;FOLD ARCOFF WDAT2 LIN P4 CPDAT2 Tool[1]:cmttorch Base[1]:vrashatel ;%{PE}
  ;FOLD Parameters ;%{h}
    ;Params IlfProvider=kukaroboter.arctech.arcofflin; Kuka.IsGlobalPoint=False; Kuka.PointName=P4; Kuka.BlendingEnabled=False; Kuka.MoveDataName=CPDAT2; Kuka.VelocityPath=0.01; Kuka.CurrentCDSetIndex=0; Kuka.MovementParameterFieldEnabled=True; ArcTech.WdatVarName=WDAT2; ArcTech.Basic=3.4.3.1264
  ;ENDFOLD
  $BWDSTART = FALSE
  LDAT_ACT = LCPDAT2
  FDAT_ACT = FP4
  BAS(#CP_PARAMS, gArcBasVelDefinition)
  SET_CD_PARAMS (0)
  TRIGGER WHEN PATH = ArcGetPath(#ArcOffBefore, WDAT2) DELAY = 0 DO ArcMainNG(#ArcOffBeforeOffStd, WDAT2, WP4) PRIO = -1
  TRIGGER WHEN PATH = ArcGetPath(#OnTheFlyArcOff, WDAT2) DELAY = 0 DO ArcMainNG(#ArcOffMoveStd, WDAT2, WP4) PRIO = -1
  ArcMainNG(#ArcOffBeforeMoveStd, WDAT2, WP4)
  LIN XP4
  ArcMainNG(#ArcOffAfterMoveStd, WDAT2, WP4)
;ENDFOLD
   $VEL.CP = 0.080
   LIN  {X -8.829, Y -3.738, Z 19.500, A 0.000, B 0.000, C 0.000} C_DIS

;FOLD ARCON WDAT1 LIN P3 Vel=0.5 m/s CPDAT1 Tool[1]:cmttorch Base[1]:vrashatel ;%{PE}
  ;FOLD Parameters ;%{h}
    ;Params IlfProvider=kukaroboter.arctech.arconlin; Kuka.IsGlobalPoint=False; Kuka.PointName=P3; Kuka.BlendingEnabled=False; Kuka.MoveDataName=CPDAT1; Kuka.VelocityPath=0.5; Kuka.CurrentCDSetIndex=0; Kuka.MovementParameterFieldEnabled=True; ArcTech.WdatVarName=WDAT1; ArcTech.Basic=3.4.3.1264
  ;ENDFOLD
  $BWDSTART = FALSE
  LDAT_ACT = LCPDAT1
  FDAT_ACT = FP3
  BAS(#CP_PARAMS, 0.5)
  SET_CD_PARAMS (0)
  TRIGGER WHEN DISTANCE = 1 DELAY = ArcGetDelay(#PreDefinition, WDAT1) DO ArcMainNG(#PreDefinition, WDAT1, WP3) PRIO = -1
  TRIGGER WHEN PATH = ArcGetPath(#OnTheFlyArcOn, WDAT1) DELAY = ArcGetDelay(#GasPreflow, WDAT1) DO ArcMainNG(#GasPreflow, WDAT1, WP3) PRIO = -1
  TRIGGER WHEN PATH = ArcGetPath(#OnTheFlyArcOn, WDAT1) DELAY = 0 DO ArcMainNG(#ArcOnMoveStd, WDAT1, WP3) PRIO = -1
  ArcMainNG(#ArcOnBeforeMoveStd, WDAT1, WP3)
  LIN XP3
  ArcMainNG(#ArcOnAfterMoveStd, WDAT1, WP3)
;ENDFOLD
   $VEL.CP = 0.060
   LIN  {X -1.457, Y 3.633, Z 19.500, A 0.000, B 0.000, C 0.000} C_DIS

;FOLD ARCOFF WDAT2 LIN P4 CPDAT2 Tool[1]:cmttorch Base[1]:vrashatel ;%{PE}
  ;FOLD Parameters ;%{h}
    ;Params IlfProvider=kukaroboter.arctech.arcofflin; Kuka.IsGlobalPoint=False; Kuka.PointName=P4; Kuka.BlendingEnabled=False; Kuka.MoveDataName=CPDAT2; Kuka.VelocityPath=0.01; Kuka.CurrentCDSetIndex=0; Kuka.MovementParameterFieldEnabled=True; ArcTech.WdatVarName=WDAT2; ArcTech.Basic=3.4.3.1264
  ;ENDFOLD
  $BWDSTART = FALSE
  LDAT_ACT = LCPDAT2
  FDAT_ACT = FP4
  BAS(#CP_PARAMS, gArcBasVelDefinition)
  SET_CD_PARAMS (0)
  TRIGGER WHEN PATH = ArcGetPath(#ArcOffBefore, WDAT2) DELAY = 0 DO ArcMainNG(#ArcOffBeforeOffStd, WDAT2, WP4) PRIO = -1
  TRIGGER WHEN PATH = ArcGetPath(#OnTheFlyArcOff, WDAT2) DELAY = 0 DO ArcMainNG(#ArcOffMoveStd, WDAT2, WP4) PRIO = -1
  ArcMainNG(#ArcOffBeforeMoveStd, WDAT2, WP4)
  LIN XP4
  ArcMainNG(#ArcOffAfterMoveStd, WDAT2, WP4)
;ENDFOLD
   $VEL.CP = 0.080
   LIN  {X -2.023, Y 3.633, Z 19.500, A 0.000, B 0.000, C 0.000} C_DIS

;FOLD ARCON WDAT1 LIN P3 Vel=0.5 m/s CPDAT1 Tool[1]:cmttorch Base[1]:vrashatel ;%{PE}
  ;FOLD Parameters ;%{h}
    ;Params IlfProvider=kukaroboter.arctech.arconlin; Kuka.IsGlobalPoint=False; Kuka.PointName=P3; Kuka.BlendingEnabled=False; Kuka.MoveDataName=CPDAT1; Kuka.VelocityPath=0.5; Kuka.CurrentCDSetIndex=0; Kuka.MovementParameterFieldEnabled=True; ArcTech.WdatVarName=WDAT1; ArcTech.Basic=3.4.3.1264
  ;ENDFOLD
  $BWDSTART = FALSE
  LDAT_ACT = LCPDAT1
  FDAT_ACT = FP3
  BAS(#CP_PARAMS, 0.5)
  SET_CD_PARAMS (0)
  TRIGGER WHEN DISTANCE = 1 DELAY = ArcGetDelay(#PreDefinition, WDAT1) DO ArcMainNG(#PreDefinition, WDAT1, WP3) PRIO = -1
  TRIGGER WHEN PATH = ArcGetPath(#OnTheFlyArcOn, WDAT1) DELAY = ArcGetDelay(#GasPreflow, WDAT1) DO ArcMainNG(#GasPreflow, WDAT1, WP3) PRIO = -1
  TRIGGER WHEN PATH = ArcGetPath(#OnTheFlyArcOn, WDAT1) DELAY = 0 DO ArcMainNG(#ArcOnMoveStd, WDAT1, WP3) PRIO = -1
  ArcMainNG(#ArcOnBeforeMoveStd, WDAT1, WP3)
  LIN XP3
  ArcMainNG(#ArcOnAfterMoveStd, WDAT1, WP3)
;ENDFOLD
   $VEL.CP = 0.060
   LIN  {X -8.829, Y -3.172, Z 19.500, A 0.000, B 0.000, C 0.000} C_DIS

;FOLD ARCOFF WDAT2 LIN P4 CPDAT2 Tool[1]:cmttorch Base[1]:vrashatel ;%{PE}
  ;FOLD Parameters ;%{h}
    ;Params IlfProvider=kukaroboter.arctech.arcofflin; Kuka.IsGlobalPoint=False; Kuka.PointName=P4; Kuka.BlendingEnabled=False; Kuka.MoveDataName=CPDAT2; Kuka.VelocityPath=0.01; Kuka.CurrentCDSetIndex=0; Kuka.MovementParameterFieldEnabled=True; ArcTech.WdatVarName=WDAT2; ArcTech.Basic=3.4.3.1264
  ;ENDFOLD
  $BWDSTART = FALSE
  LDAT_ACT = LCPDAT2
  FDAT_ACT = FP4
  BAS(#CP_PARAMS, gArcBasVelDefinition)
  SET_CD_PARAMS (0)
  TRIGGER WHEN PATH = ArcGetPath(#ArcOffBefore, WDAT2) DELAY = 0 DO ArcMainNG(#ArcOffBeforeOffStd, WDAT2, WP4) PRIO = -1
  TRIGGER WHEN PATH = ArcGetPath(#OnTheFlyArcOff, WDAT2) DELAY = 0 DO ArcMainNG(#ArcOffMoveStd, WDAT2, WP4) PRIO = -1
  ArcMainNG(#ArcOffBeforeMoveStd, WDAT2, WP4)
  LIN XP4
  ArcMainNG(#ArcOffAfterMoveStd, WDAT2, WP4)
;ENDFOLD
   $VEL.CP = 0.080
   LIN  {X -8.829, Y -2.607, Z 19.500, A 0.000, B 0.000, C 0.000} C_DIS

;FOLD ARCON WDAT1 LIN P3 Vel=0.5 m/s CPDAT1 Tool[1]:cmttorch Base[1]:vrashatel ;%{PE}
  ;FOLD Parameters ;%{h}
    ;Params IlfProvider=kukaroboter.arctech.arconlin; Kuka.IsGlobalPoint=False; Kuka.PointName=P3; Kuka.BlendingEnabled=False; Kuka.MoveDataName=CPDAT1; Kuka.VelocityPath=0.5; Kuka.CurrentCDSetIndex=0; Kuka.MovementParameterFieldEnabled=True; ArcTech.WdatVarName=WDAT1; ArcTech.Basic=3.4.3.1264
  ;ENDFOLD
  $BWDSTART = FALSE
  LDAT_ACT = LCPDAT1
  FDAT_ACT = FP3
  BAS(#CP_PARAMS, 0.5)
  SET_CD_PARAMS (0)
  TRIGGER WHEN DISTANCE = 1 DELAY = ArcGetDelay(#PreDefinition, WDAT1) DO ArcMainNG(#PreDefinition, WDAT1, WP3) PRIO = -1
  TRIGGER WHEN PATH = ArcGetPath(#OnTheFlyArcOn, WDAT1) DELAY = ArcGetDelay(#GasPreflow, WDAT1) DO ArcMainNG(#GasPreflow, WDAT1, WP3) PRIO = -1
  TRIGGER WHEN PATH = ArcGetPath(#OnTheFlyArcOn, WDAT1) DELAY = 0 DO ArcMainNG(#ArcOnMoveStd, WDAT1, WP3) PRIO = -1
  ArcMainNG(#ArcOnBeforeMoveStd, WDAT1, WP3)
  LIN XP3
  ArcMainNG(#ArcOnAfterMoveStd, WDAT1, WP3)
;ENDFOLD
   $VEL.CP = 0.060
   LIN  {X -2.588, Y 3.633, Z 19.500, A 0.000, B 0.000, C 0.000} C_DIS

;FOLD ARCOFF WDAT2 LIN P4 CPDAT2 Tool[1]:cmttorch Base[1]:vrashatel ;%{PE}
  ;FOLD Parameters ;%{h}
    ;Params IlfProvider=kukaroboter.arctech.arcofflin; Kuka.IsGlobalPoint=False; Kuka.PointName=P4; Kuka.BlendingEnabled=False; Kuka.MoveDataName=CPDAT2; Kuka.VelocityPath=0.01; Kuka.CurrentCDSetIndex=0; Kuka.MovementParameterFieldEnabled=True; ArcTech.WdatVarName=WDAT2; ArcTech.Basic=3.4.3.1264
  ;ENDFOLD
  $BWDSTART = FALSE
  LDAT_ACT = LCPDAT2
  FDAT_ACT = FP4
  BAS(#CP_PARAMS, gArcBasVelDefinition)
  SET_CD_PARAMS (0)
  TRIGGER WHEN PATH = ArcGetPath(#ArcOffBefore, WDAT2) DELAY = 0 DO ArcMainNG(#ArcOffBeforeOffStd, WDAT2, WP4) PRIO = -1
  TRIGGER WHEN PATH = ArcGetPath(#OnTheFlyArcOff, WDAT2) DELAY = 0 DO ArcMainNG(#ArcOffMoveStd, WDAT2, WP4) PRIO = -1
  ArcMainNG(#ArcOffBeforeMoveStd, WDAT2, WP4)
  LIN XP4
  ArcMainNG(#ArcOffAfterMoveStd, WDAT2, WP4)
;ENDFOLD
   $VEL.CP = 0.080
   LIN  {X -3.154, Y 3.633, Z 19.500, A 0.000, B 0.000, C 0.000} C_DIS

;FOLD ARCON WDAT1 LIN P3 Vel=0.5 m/s CPDAT1 Tool[1]:cmttorch Base[1]:vrashatel ;%{PE}
  ;FOLD Parameters ;%{h}
    ;Params IlfProvider=kukaroboter.arctech.arconlin; Kuka.IsGlobalPoint=False; Kuka.PointName=P3; Kuka.BlendingEnabled=False; Kuka.MoveDataName=CPDAT1; Kuka.VelocityPath=0.5; Kuka.CurrentCDSetIndex=0; Kuka.MovementParameterFieldEnabled=True; ArcTech.WdatVarName=WDAT1; ArcTech.Basic=3.4.3.1264
  ;ENDFOLD
  $BWDSTART = FALSE
  LDAT_ACT = LCPDAT1
  FDAT_ACT = FP3
  BAS(#CP_PARAMS, 0.5)
  SET_CD_PARAMS (0)
  TRIGGER WHEN DISTANCE = 1 DELAY = ArcGetDelay(#PreDefinition, WDAT1) DO ArcMainNG(#PreDefinition, WDAT1, WP3) PRIO = -1
  TRIGGER WHEN PATH = ArcGetPath(#OnTheFlyArcOn, WDAT1) DELAY = ArcGetDelay(#GasPreflow, WDAT1) DO ArcMainNG(#GasPreflow, WDAT1, WP3) PRIO = -1
  TRIGGER WHEN PATH = ArcGetPath(#OnTheFlyArcOn, WDAT1) DELAY = 0 DO ArcMainNG(#ArcOnMoveStd, WDAT1, WP3) PRIO = -1
  ArcMainNG(#ArcOnBeforeMoveStd, WDAT1, WP3)
  LIN XP3
  ArcMainNG(#ArcOnAfterMoveStd, WDAT1, WP3)
;ENDFOLD
   $VEL.CP = 0.060
   LIN  {X -8.829, Y -2.041, Z 19.500, A 0.000, B 0.000, C 0.000} C_DIS

;FOLD ARCOFF WDAT2 LIN P4 CPDAT2 Tool[1]:cmttorch Base[1]:vrashatel ;%{PE}
  ;FOLD Parameters ;%{h}
    ;Params IlfProvider=kukaroboter.arctech.arcofflin; Kuka.IsGlobalPoint=False; Kuka.PointName=P4; Kuka.BlendingEnabled=False; Kuka.MoveDataName=CPDAT2; Kuka.VelocityPath=0.01; Kuka.CurrentCDSetIndex=0; Kuka.MovementParameterFieldEnabled=True; ArcTech.WdatVarName=WDAT2; ArcTech.Basic=3.4.3.1264
  ;ENDFOLD
  $BWDSTART = FALSE
  LDAT_ACT = LCPDAT2
  FDAT_ACT = FP4
  BAS(#CP_PARAMS, gArcBasVelDefinition)
  SET_CD_PARAMS (0)
  TRIGGER WHEN PATH = ArcGetPath(#ArcOffBefore, WDAT2) DELAY = 0 DO ArcMainNG(#ArcOffBeforeOffStd, WDAT2, WP4) PRIO = -1
  TRIGGER WHEN PATH = ArcGetPath(#OnTheFlyArcOff, WDAT2) DELAY = 0 DO ArcMainNG(#ArcOffMoveStd, WDAT2, WP4) PRIO = -1
  ArcMainNG(#ArcOffBeforeMoveStd, WDAT2, WP4)
  LIN XP4
  ArcMainNG(#ArcOffAfterMoveStd, WDAT2, WP4)
;ENDFOLD
   $VEL.CP = 0.080
   LIN  {X -8.829, Y -1.475, Z 19.500, A 0.000, B 0.000, C 0.000} C_DIS

;FOLD ARCON WDAT1 LIN P3 Vel=0.5 m/s CPDAT1 Tool[1]:cmttorch Base[1]:vrashatel ;%{PE}
  ;FOLD Parameters ;%{h}
    ;Params IlfProvider=kukaroboter.arctech.arconlin; Kuka.IsGlobalPoint=False; Kuka.PointName=P3; Kuka.BlendingEnabled=False; Kuka.MoveDataName=CPDAT1; Kuka.VelocityPath=0.5; Kuka.CurrentCDSetIndex=0; Kuka.MovementParameterFieldEnabled=True; ArcTech.WdatVarName=WDAT1; ArcTech.Basic=3.4.3.1264
  ;ENDFOLD
  $BWDSTART = FALSE
  LDAT_ACT = LCPDAT1
  FDAT_ACT = FP3
  BAS(#CP_PARAMS, 0.5)
  SET_CD_PARAMS (0)
  TRIGGER WHEN DISTANCE = 1 DELAY = ArcGetDelay(#PreDefinition, WDAT1) DO ArcMainNG(#PreDefinition, WDAT1, WP3) PRIO = -1
  TRIGGER WHEN PATH = ArcGetPath(#OnTheFlyArcOn, WDAT1) DELAY = ArcGetDelay(#GasPreflow, WDAT1) DO ArcMainNG(#GasPreflow, WDAT1, WP3) PRIO = -1
  TRIGGER WHEN PATH = ArcGetPath(#OnTheFlyArcOn, WDAT1) DELAY = 0 DO ArcMainNG(#ArcOnMoveStd, WDAT1, WP3) PRIO = -1
  ArcMainNG(#ArcOnBeforeMoveStd, WDAT1, WP3)
  LIN XP3
  ArcMainNG(#ArcOnAfterMoveStd, WDAT1, WP3)
;ENDFOLD
   $VEL.CP = 0.060
   LIN  {X -3.720, Y 3.633, Z 19.500, A 0.000, B 0.000, C 0.000} C_DIS

;FOLD ARCOFF WDAT2 LIN P4 CPDAT2 Tool[1]:cmttorch Base[1]:vrashatel ;%{PE}
  ;FOLD Parameters ;%{h}
    ;Params IlfProvider=kukaroboter.arctech.arcofflin; Kuka.IsGlobalPoint=False; Kuka.PointName=P4; Kuka.BlendingEnabled=False; Kuka.MoveDataName=CPDAT2; Kuka.VelocityPath=0.01; Kuka.CurrentCDSetIndex=0; Kuka.MovementParameterFieldEnabled=True; ArcTech.WdatVarName=WDAT2; ArcTech.Basic=3.4.3.1264
  ;ENDFOLD
  $BWDSTART = FALSE
  LDAT_ACT = LCPDAT2
  FDAT_ACT = FP4
  BAS(#CP_PARAMS, gArcBasVelDefinition)
  SET_CD_PARAMS (0)
  TRIGGER WHEN PATH = ArcGetPath(#ArcOffBefore, WDAT2) DELAY = 0 DO ArcMainNG(#ArcOffBeforeOffStd, WDAT2, WP4) PRIO = -1
  TRIGGER WHEN PATH = ArcGetPath(#OnTheFlyArcOff, WDAT2) DELAY = 0 DO ArcMainNG(#ArcOffMoveStd, WDAT2, WP4) PRIO = -1
  ArcMainNG(#ArcOffBeforeMoveStd, WDAT2, WP4)
  LIN XP4
  ArcMainNG(#ArcOffAfterMoveStd, WDAT2, WP4)
;ENDFOLD
   $VEL.CP = 0.080
   LIN  {X -4.285, Y 3.633, Z 19.500, A 0.000, B 0.000, C 0.000} C_DIS

;FOLD ARCON WDAT1 LIN P3 Vel=0.5 m/s CPDAT1 Tool[1]:cmttorch Base[1]:vrashatel ;%{PE}
  ;FOLD Parameters ;%{h}
    ;Params IlfProvider=kukaroboter.arctech.arconlin; Kuka.IsGlobalPoint=False; Kuka.PointName=P3; Kuka.BlendingEnabled=False; Kuka.MoveDataName=CPDAT1; Kuka.VelocityPath=0.5; Kuka.CurrentCDSetIndex=0; Kuka.MovementParameterFieldEnabled=True; ArcTech.WdatVarName=WDAT1; ArcTech.Basic=3.4.3.1264
  ;ENDFOLD
  $BWDSTART = FALSE
  LDAT_ACT = LCPDAT1
  FDAT_ACT = FP3
  BAS(#CP_PARAMS, 0.5)
  SET_CD_PARAMS (0)
  TRIGGER WHEN DISTANCE = 1 DELAY = ArcGetDelay(#PreDefinition, WDAT1) DO ArcMainNG(#PreDefinition, WDAT1, WP3) PRIO = -1
  TRIGGER WHEN PATH = ArcGetPath(#OnTheFlyArcOn, WDAT1) DELAY = ArcGetDelay(#GasPreflow, WDAT1) DO ArcMainNG(#GasPreflow, WDAT1, WP3) PRIO = -1
  TRIGGER WHEN PATH = ArcGetPath(#OnTheFlyArcOn, WDAT1) DELAY = 0 DO ArcMainNG(#ArcOnMoveStd, WDAT1, WP3) PRIO = -1
  ArcMainNG(#ArcOnBeforeMoveStd, WDAT1, WP3)
  LIN XP3
  ArcMainNG(#ArcOnAfterMoveStd, WDAT1, WP3)
;ENDFOLD
   $VEL.CP = 0.060
   LIN  {X -8.829, Y -0.910, Z 19.500, A 0.000, B 0.000, C 0.000} C_DIS

;FOLD ARCOFF WDAT2 LIN P4 CPDAT2 Tool[1]:cmttorch Base[1]:vrashatel ;%{PE}
  ;FOLD Parameters ;%{h}
    ;Params IlfProvider=kukaroboter.arctech.arcofflin; Kuka.IsGlobalPoint=False; Kuka.PointName=P4; Kuka.BlendingEnabled=False; Kuka.MoveDataName=CPDAT2; Kuka.VelocityPath=0.01; Kuka.CurrentCDSetIndex=0; Kuka.MovementParameterFieldEnabled=True; ArcTech.WdatVarName=WDAT2; ArcTech.Basic=3.4.3.1264
  ;ENDFOLD
  $BWDSTART = FALSE
  LDAT_ACT = LCPDAT2
  FDAT_ACT = FP4
  BAS(#CP_PARAMS, gArcBasVelDefinition)
  SET_CD_PARAMS (0)
  TRIGGER WHEN PATH = ArcGetPath(#ArcOffBefore, WDAT2) DELAY = 0 DO ArcMainNG(#ArcOffBeforeOffStd, WDAT2, WP4) PRIO = -1
  TRIGGER WHEN PATH = ArcGetPath(#OnTheFlyArcOff, WDAT2) DELAY = 0 DO ArcMainNG(#ArcOffMoveStd, WDAT2, WP4) PRIO = -1
  ArcMainNG(#ArcOffBeforeMoveStd, WDAT2, WP4)
  LIN XP4
  ArcMainNG(#ArcOffAfterMoveStd, WDAT2, WP4)
;ENDFOLD
   $VEL.CP = 0.080
   LIN  {X -8.829, Y -0.344, Z 19.500, A 0.000, B 0.000, C 0.000} C_DIS

;FOLD ARCON WDAT1 LIN P3 Vel=0.5 m/s CPDAT1 Tool[1]:cmttorch Base[1]:vrashatel ;%{PE}
  ;FOLD Parameters ;%{h}
    ;Params IlfProvider=kukaroboter.arctech.arconlin; Kuka.IsGlobalPoint=False; Kuka.PointName=P3; Kuka.BlendingEnabled=False; Kuka.MoveDataName=CPDAT1; Kuka.VelocityPath=0.5; Kuka.CurrentCDSetIndex=0; Kuka.MovementParameterFieldEnabled=True; ArcTech.WdatVarName=WDAT1; ArcTech.Basic=3.4.3.1264
  ;ENDFOLD
  $BWDSTART = FALSE
  LDAT_ACT = LCPDAT1
  FDAT_ACT = FP3
  BAS(#CP_PARAMS, 0.5)
  SET_CD_PARAMS (0)
  TRIGGER WHEN DISTANCE = 1 DELAY = ArcGetDelay(#PreDefinition, WDAT1) DO ArcMainNG(#PreDefinition, WDAT1, WP3) PRIO = -1
  TRIGGER WHEN PATH = ArcGetPath(#OnTheFlyArcOn, WDAT1) DELAY = ArcGetDelay(#GasPreflow, WDAT1) DO ArcMainNG(#GasPreflow, WDAT1, WP3) PRIO = -1
  TRIGGER WHEN PATH = ArcGetPath(#OnTheFlyArcOn, WDAT1) DELAY = 0 DO ArcMainNG(#ArcOnMoveStd, WDAT1, WP3) PRIO = -1
  ArcMainNG(#ArcOnBeforeMoveStd, WDAT1, WP3)
  LIN XP3
  ArcMainNG(#ArcOnAfterMoveStd, WDAT1, WP3)
;ENDFOLD
   $VEL.CP = 0.060
   LIN  {X -4.763, Y 3.722, Z 19.500, A 0.000, B 0.000, C 0.000} C_DIS

;FOLD ARCOFF WDAT2 LIN P4 CPDAT2 Tool[1]:cmttorch Base[1]:vrashatel ;%{PE}
  ;FOLD Parameters ;%{h}
    ;Params IlfProvider=kukaroboter.arctech.arcofflin; Kuka.IsGlobalPoint=False; Kuka.PointName=P4; Kuka.BlendingEnabled=False; Kuka.MoveDataName=CPDAT2; Kuka.VelocityPath=0.01; Kuka.CurrentCDSetIndex=0; Kuka.MovementParameterFieldEnabled=True; ArcTech.WdatVarName=WDAT2; ArcTech.Basic=3.4.3.1264
  ;ENDFOLD
  $BWDSTART = FALSE
  LDAT_ACT = LCPDAT2
  FDAT_ACT = FP4
  BAS(#CP_PARAMS, gArcBasVelDefinition)
  SET_CD_PARAMS (0)
  TRIGGER WHEN PATH = ArcGetPath(#ArcOffBefore, WDAT2) DELAY = 0 DO ArcMainNG(#ArcOffBeforeOffStd, WDAT2, WP4) PRIO = -1
  TRIGGER WHEN PATH = ArcGetPath(#OnTheFlyArcOff, WDAT2) DELAY = 0 DO ArcMainNG(#ArcOffMoveStd, WDAT2, WP4) PRIO = -1
  ArcMainNG(#ArcOffBeforeMoveStd, WDAT2, WP4)
  LIN XP4
  ArcMainNG(#ArcOffAfterMoveStd, WDAT2, WP4)
;ENDFOLD
   $VEL.CP = 0.080
   LIN  {X -4.763, Y 4.287, Z 19.500, A 0.000, B 0.000, C 0.000} C_DIS

;FOLD ARCON WDAT1 LIN P3 Vel=0.5 m/s CPDAT1 Tool[1]:cmttorch Base[1]:vrashatel ;%{PE}
  ;FOLD Parameters ;%{h}
    ;Params IlfProvider=kukaroboter.arctech.arconlin; Kuka.IsGlobalPoint=False; Kuka.PointName=P3; Kuka.BlendingEnabled=False; Kuka.MoveDataName=CPDAT1; Kuka.VelocityPath=0.5; Kuka.CurrentCDSetIndex=0; Kuka.MovementParameterFieldEnabled=True; ArcTech.WdatVarName=WDAT1; ArcTech.Basic=3.4.3.1264
  ;ENDFOLD
  $BWDSTART = FALSE
  LDAT_ACT = LCPDAT1
  FDAT_ACT = FP3
  BAS(#CP_PARAMS, 0.5)
  SET_CD_PARAMS (0)
  TRIGGER WHEN DISTANCE = 1 DELAY = ArcGetDelay(#PreDefinition, WDAT1) DO ArcMainNG(#PreDefinition, WDAT1, WP3) PRIO = -1
  TRIGGER WHEN PATH = ArcGetPath(#OnTheFlyArcOn, WDAT1) DELAY = ArcGetDelay(#GasPreflow, WDAT1) DO ArcMainNG(#GasPreflow, WDAT1, WP3) PRIO = -1
  TRIGGER WHEN PATH = ArcGetPath(#OnTheFlyArcOn, WDAT1) DELAY = 0 DO ArcMainNG(#ArcOnMoveStd, WDAT1, WP3) PRIO = -1
  ArcMainNG(#ArcOnBeforeMoveStd, WDAT1, WP3)
  LIN XP3
  ArcMainNG(#ArcOnAfterMoveStd, WDAT1, WP3)
;ENDFOLD
   $VEL.CP = 0.060
   LIN  {X -8.829, Y 0.221, Z 19.500, A 0.000, B 0.000, C 0.000} C_DIS

;FOLD ARCOFF WDAT2 LIN P4 CPDAT2 Tool[1]:cmttorch Base[1]:vrashatel ;%{PE}
  ;FOLD Parameters ;%{h}
    ;Params IlfProvider=kukaroboter.arctech.arcofflin; Kuka.IsGlobalPoint=False; Kuka.PointName=P4; Kuka.BlendingEnabled=False; Kuka.MoveDataName=CPDAT2; Kuka.VelocityPath=0.01; Kuka.CurrentCDSetIndex=0; Kuka.MovementParameterFieldEnabled=True; ArcTech.WdatVarName=WDAT2; ArcTech.Basic=3.4.3.1264
  ;ENDFOLD
  $BWDSTART = FALSE
  LDAT_ACT = LCPDAT2
  FDAT_ACT = FP4
  BAS(#CP_PARAMS, gArcBasVelDefinition)
  SET_CD_PARAMS (0)
  TRIGGER WHEN PATH = ArcGetPath(#ArcOffBefore, WDAT2) DELAY = 0 DO ArcMainNG(#ArcOffBeforeOffStd, WDAT2, WP4) PRIO = -1
  TRIGGER WHEN PATH = ArcGetPath(#OnTheFlyArcOff, WDAT2) DELAY = 0 DO ArcMainNG(#ArcOffMoveStd, WDAT2, WP4) PRIO = -1
  ArcMainNG(#ArcOffBeforeMoveStd, WDAT2, WP4)
  LIN XP4
  ArcMainNG(#ArcOffAfterMoveStd, WDAT2, WP4)
;ENDFOLD
   $VEL.CP = 0.080
   LIN  {X -8.829, Y 0.787, Z 19.500, A 0.000, B 0.000, C 0.000} C_DIS

;FOLD ARCON WDAT1 LIN P3 Vel=0.5 m/s CPDAT1 Tool[1]:cmttorch Base[1]:vrashatel ;%{PE}
  ;FOLD Parameters ;%{h}
    ;Params IlfProvider=kukaroboter.arctech.arconlin; Kuka.IsGlobalPoint=False; Kuka.PointName=P3; Kuka.BlendingEnabled=False; Kuka.MoveDataName=CPDAT1; Kuka.VelocityPath=0.5; Kuka.CurrentCDSetIndex=0; Kuka.MovementParameterFieldEnabled=True; ArcTech.WdatVarName=WDAT1; ArcTech.Basic=3.4.3.1264
  ;ENDFOLD
  $BWDSTART = FALSE
  LDAT_ACT = LCPDAT1
  FDAT_ACT = FP3
  BAS(#CP_PARAMS, 0.5)
  SET_CD_PARAMS (0)
  TRIGGER WHEN DISTANCE = 1 DELAY = ArcGetDelay(#PreDefinition, WDAT1) DO ArcMainNG(#PreDefinition, WDAT1, WP3) PRIO = -1
  TRIGGER WHEN PATH = ArcGetPath(#OnTheFlyArcOn, WDAT1) DELAY = ArcGetDelay(#GasPreflow, WDAT1) DO ArcMainNG(#GasPreflow, WDAT1, WP3) PRIO = -1
  TRIGGER WHEN PATH = ArcGetPath(#OnTheFlyArcOn, WDAT1) DELAY = 0 DO ArcMainNG(#ArcOnMoveStd, WDAT1, WP3) PRIO = -1
  ArcMainNG(#ArcOnBeforeMoveStd, WDAT1, WP3)
  LIN XP3
  ArcMainNG(#ArcOnAfterMoveStd, WDAT1, WP3)
;ENDFOLD
   $VEL.CP = 0.060
   LIN  {X -4.763, Y 4.853, Z 19.500, A 0.000, B 0.000, C 0.000} C_DIS

;FOLD ARCOFF WDAT2 LIN P4 CPDAT2 Tool[1]:cmttorch Base[1]:vrashatel ;%{PE}
  ;FOLD Parameters ;%{h}
    ;Params IlfProvider=kukaroboter.arctech.arcofflin; Kuka.IsGlobalPoint=False; Kuka.PointName=P4; Kuka.BlendingEnabled=False; Kuka.MoveDataName=CPDAT2; Kuka.VelocityPath=0.01; Kuka.CurrentCDSetIndex=0; Kuka.MovementParameterFieldEnabled=True; ArcTech.WdatVarName=WDAT2; ArcTech.Basic=3.4.3.1264
  ;ENDFOLD
  $BWDSTART = FALSE
  LDAT_ACT = LCPDAT2
  FDAT_ACT = FP4
  BAS(#CP_PARAMS, gArcBasVelDefinition)
  SET_CD_PARAMS (0)
  TRIGGER WHEN PATH = ArcGetPath(#ArcOffBefore, WDAT2) DELAY = 0 DO ArcMainNG(#ArcOffBeforeOffStd, WDAT2, WP4) PRIO = -1
  TRIGGER WHEN PATH = ArcGetPath(#OnTheFlyArcOff, WDAT2) DELAY = 0 DO ArcMainNG(#ArcOffMoveStd, WDAT2, WP4) PRIO = -1
  ArcMainNG(#ArcOffBeforeMoveStd, WDAT2, WP4)
  LIN XP4
  ArcMainNG(#ArcOffAfterMoveStd, WDAT2, WP4)
;ENDFOLD
   $VEL.CP = 0.080
   LIN  {X -4.763, Y 5.419, Z 19.500, A 0.000, B 0.000, C 0.000} C_DIS

;FOLD ARCON WDAT1 LIN P3 Vel=0.5 m/s CPDAT1 Tool[1]:cmttorch Base[1]:vrashatel ;%{PE}
  ;FOLD Parameters ;%{h}
    ;Params IlfProvider=kukaroboter.arctech.arconlin; Kuka.IsGlobalPoint=False; Kuka.PointName=P3; Kuka.BlendingEnabled=False; Kuka.MoveDataName=CPDAT1; Kuka.VelocityPath=0.5; Kuka.CurrentCDSetIndex=0; Kuka.MovementParameterFieldEnabled=True; ArcTech.WdatVarName=WDAT1; ArcTech.Basic=3.4.3.1264
  ;ENDFOLD
  $BWDSTART = FALSE
  LDAT_ACT = LCPDAT1
  FDAT_ACT = FP3
  BAS(#CP_PARAMS, 0.5)
  SET_CD_PARAMS (0)
  TRIGGER WHEN DISTANCE = 1 DELAY = ArcGetDelay(#PreDefinition, WDAT1) DO ArcMainNG(#PreDefinition, WDAT1, WP3) PRIO = -1
  TRIGGER WHEN PATH = ArcGetPath(#OnTheFlyArcOn, WDAT1) DELAY = ArcGetDelay(#GasPreflow, WDAT1) DO ArcMainNG(#GasPreflow, WDAT1, WP3) PRIO = -1
  TRIGGER WHEN PATH = ArcGetPath(#OnTheFlyArcOn, WDAT1) DELAY = 0 DO ArcMainNG(#ArcOnMoveStd, WDAT1, WP3) PRIO = -1
  ArcMainNG(#ArcOnBeforeMoveStd, WDAT1, WP3)
  LIN XP3
  ArcMainNG(#ArcOnAfterMoveStd, WDAT1, WP3)
;ENDFOLD
   $VEL.CP = 0.060
   LIN  {X -8.829, Y 1.352, Z 19.500, A 0.000, B 0.000, C 0.000} C_DIS

;FOLD ARCOFF WDAT2 LIN P4 CPDAT2 Tool[1]:cmttorch Base[1]:vrashatel ;%{PE}
  ;FOLD Parameters ;%{h}
    ;Params IlfProvider=kukaroboter.arctech.arcofflin; Kuka.IsGlobalPoint=False; Kuka.PointName=P4; Kuka.BlendingEnabled=False; Kuka.MoveDataName=CPDAT2; Kuka.VelocityPath=0.01; Kuka.CurrentCDSetIndex=0; Kuka.MovementParameterFieldEnabled=True; ArcTech.WdatVarName=WDAT2; ArcTech.Basic=3.4.3.1264
  ;ENDFOLD
  $BWDSTART = FALSE
  LDAT_ACT = LCPDAT2
  FDAT_ACT = FP4
  BAS(#CP_PARAMS, gArcBasVelDefinition)
  SET_CD_PARAMS (0)
  TRIGGER WHEN PATH = ArcGetPath(#ArcOffBefore, WDAT2) DELAY = 0 DO ArcMainNG(#ArcOffBeforeOffStd, WDAT2, WP4) PRIO = -1
  TRIGGER WHEN PATH = ArcGetPath(#OnTheFlyArcOff, WDAT2) DELAY = 0 DO ArcMainNG(#ArcOffMoveStd, WDAT2, WP4) PRIO = -1
  ArcMainNG(#ArcOffBeforeMoveStd, WDAT2, WP4)
  LIN XP4
  ArcMainNG(#ArcOffAfterMoveStd, WDAT2, WP4)
;ENDFOLD
   $VEL.CP = 0.080
   LIN  {X -8.829, Y 1.918, Z 19.500, A 0.000, B 0.000, C 0.000} C_DIS

;FOLD ARCON WDAT1 LIN P3 Vel=0.5 m/s CPDAT1 Tool[1]:cmttorch Base[1]:vrashatel ;%{PE}
  ;FOLD Parameters ;%{h}
    ;Params IlfProvider=kukaroboter.arctech.arconlin; Kuka.IsGlobalPoint=False; Kuka.PointName=P3; Kuka.BlendingEnabled=False; Kuka.MoveDataName=CPDAT1; Kuka.VelocityPath=0.5; Kuka.CurrentCDSetIndex=0; Kuka.MovementParameterFieldEnabled=True; ArcTech.WdatVarName=WDAT1; ArcTech.Basic=3.4.3.1264
  ;ENDFOLD
  $BWDSTART = FALSE
  LDAT_ACT = LCPDAT1
  FDAT_ACT = FP3
  BAS(#CP_PARAMS, 0.5)
  SET_CD_PARAMS (0)
  TRIGGER WHEN DISTANCE = 1 DELAY = ArcGetDelay(#PreDefinition, WDAT1) DO ArcMainNG(#PreDefinition, WDAT1, WP3) PRIO = -1
  TRIGGER WHEN PATH = ArcGetPath(#OnTheFlyArcOn, WDAT1) DELAY = ArcGetDelay(#GasPreflow, WDAT1) DO ArcMainNG(#GasPreflow, WDAT1, WP3) PRIO = -1
  TRIGGER WHEN PATH = ArcGetPath(#OnTheFlyArcOn, WDAT1) DELAY = 0 DO ArcMainNG(#ArcOnMoveStd, WDAT1, WP3) PRIO = -1
  ArcMainNG(#ArcOnBeforeMoveStd, WDAT1, WP3)
  LIN XP3
  ArcMainNG(#ArcOnAfterMoveStd, WDAT1, WP3)
;ENDFOLD
   $VEL.CP = 0.060
   LIN  {X -4.763, Y 5.984, Z 19.500, A 0.000, B 0.000, C 0.000} C_DIS

;FOLD ARCOFF WDAT2 LIN P4 CPDAT2 Tool[1]:cmttorch Base[1]:vrashatel ;%{PE}
  ;FOLD Parameters ;%{h}
    ;Params IlfProvider=kukaroboter.arctech.arcofflin; Kuka.IsGlobalPoint=False; Kuka.PointName=P4; Kuka.BlendingEnabled=False; Kuka.MoveDataName=CPDAT2; Kuka.VelocityPath=0.01; Kuka.CurrentCDSetIndex=0; Kuka.MovementParameterFieldEnabled=True; ArcTech.WdatVarName=WDAT2; ArcTech.Basic=3.4.3.1264
  ;ENDFOLD
  $BWDSTART = FALSE
  LDAT_ACT = LCPDAT2
  FDAT_ACT = FP4
  BAS(#CP_PARAMS, gArcBasVelDefinition)
  SET_CD_PARAMS (0)
  TRIGGER WHEN PATH = ArcGetPath(#ArcOffBefore, WDAT2) DELAY = 0 DO ArcMainNG(#ArcOffBeforeOffStd, WDAT2, WP4) PRIO = -1
  TRIGGER WHEN PATH = ArcGetPath(#OnTheFlyArcOff, WDAT2) DELAY = 0 DO ArcMainNG(#ArcOffMoveStd, WDAT2, WP4) PRIO = -1
  ArcMainNG(#ArcOffBeforeMoveStd, WDAT2, WP4)
  LIN XP4
  ArcMainNG(#ArcOffAfterMoveStd, WDAT2, WP4)
;ENDFOLD
   $VEL.CP = 0.080
   LIN  {X -4.763, Y 6.550, Z 19.500, A 0.000, B 0.000, C 0.000} C_DIS

;FOLD ARCON WDAT1 LIN P3 Vel=0.5 m/s CPDAT1 Tool[1]:cmttorch Base[1]:vrashatel ;%{PE}
  ;FOLD Parameters ;%{h}
    ;Params IlfProvider=kukaroboter.arctech.arconlin; Kuka.IsGlobalPoint=False; Kuka.PointName=P3; Kuka.BlendingEnabled=False; Kuka.MoveDataName=CPDAT1; Kuka.VelocityPath=0.5; Kuka.CurrentCDSetIndex=0; Kuka.MovementParameterFieldEnabled=True; ArcTech.WdatVarName=WDAT1; ArcTech.Basic=3.4.3.1264
  ;ENDFOLD
  $BWDSTART = FALSE
  LDAT_ACT = LCPDAT1
  FDAT_ACT = FP3
  BAS(#CP_PARAMS, 0.5)
  SET_CD_PARAMS (0)
  TRIGGER WHEN DISTANCE = 1 DELAY = ArcGetDelay(#PreDefinition, WDAT1) DO ArcMainNG(#PreDefinition, WDAT1, WP3) PRIO = -1
  TRIGGER WHEN PATH = ArcGetPath(#OnTheFlyArcOn, WDAT1) DELAY = ArcGetDelay(#GasPreflow, WDAT1) DO ArcMainNG(#GasPreflow, WDAT1, WP3) PRIO = -1
  TRIGGER WHEN PATH = ArcGetPath(#OnTheFlyArcOn, WDAT1) DELAY = 0 DO ArcMainNG(#ArcOnMoveStd, WDAT1, WP3) PRIO = -1
  ArcMainNG(#ArcOnBeforeMoveStd, WDAT1, WP3)
  LIN XP3
  ArcMainNG(#ArcOnAfterMoveStd, WDAT1, WP3)
;ENDFOLD
   $VEL.CP = 0.060
   LIN  {X -8.829, Y 2.484, Z 19.500, A 0.000, B 0.000, C 0.000} C_DIS

;FOLD ARCOFF WDAT2 LIN P4 CPDAT2 Tool[1]:cmttorch Base[1]:vrashatel ;%{PE}
  ;FOLD Parameters ;%{h}
    ;Params IlfProvider=kukaroboter.arctech.arcofflin; Kuka.IsGlobalPoint=False; Kuka.PointName=P4; Kuka.BlendingEnabled=False; Kuka.MoveDataName=CPDAT2; Kuka.VelocityPath=0.01; Kuka.CurrentCDSetIndex=0; Kuka.MovementParameterFieldEnabled=True; ArcTech.WdatVarName=WDAT2; ArcTech.Basic=3.4.3.1264
  ;ENDFOLD
  $BWDSTART = FALSE
  LDAT_ACT = LCPDAT2
  FDAT_ACT = FP4
  BAS(#CP_PARAMS, gArcBasVelDefinition)
  SET_CD_PARAMS (0)
  TRIGGER WHEN PATH = ArcGetPath(#ArcOffBefore, WDAT2) DELAY = 0 DO ArcMainNG(#ArcOffBeforeOffStd, WDAT2, WP4) PRIO = -1
  TRIGGER WHEN PATH = ArcGetPath(#OnTheFlyArcOff, WDAT2) DELAY = 0 DO ArcMainNG(#ArcOffMoveStd, WDAT2, WP4) PRIO = -1
  ArcMainNG(#ArcOffBeforeMoveStd, WDAT2, WP4)
  LIN XP4
  ArcMainNG(#ArcOffAfterMoveStd, WDAT2, WP4)
;ENDFOLD
   $VEL.CP = 0.060
   LIN  {X -8.899, Y 2.414, Z 19.500, A 0.000, B 0.000, C 0.000} C_DIS
   $VEL.CP = 0.080
   LIN  {X -9.290, Y 2.414, Z 19.500, A 0.000, B 0.000, C 0.000} C_DIS
   $VEL.CP = 0.080
   LIN  {X -9.218, Y -9.218, Z 19.500, A 0.000, B 0.000, C 0.000} C_DIS
   $VEL.CP = 0.080
   LIN  {X 4.181, Y -9.290, Z 19.500, A 0.000, B 0.000, C 0.000} C_DIS
   $VEL.CP = 0.080
   LIN  {X 4.181, Y -8.829, Z 19.500, A 0.000, B 0.000, C 0.000} C_DIS

;FOLD ARCON WDAT1 LIN P3 Vel=0.5 m/s CPDAT1 Tool[1]:cmttorch Base[1]:vrashatel ;%{PE}
  ;FOLD Parameters ;%{h}
    ;Params IlfProvider=kukaroboter.arctech.arconlin; Kuka.IsGlobalPoint=False; Kuka.PointName=P3; Kuka.BlendingEnabled=False; Kuka.MoveDataName=CPDAT1; Kuka.VelocityPath=0.5; Kuka.CurrentCDSetIndex=0; Kuka.MovementParameterFieldEnabled=True; ArcTech.WdatVarName=WDAT1; ArcTech.Basic=3.4.3.1264
  ;ENDFOLD
  $BWDSTART = FALSE
  LDAT_ACT = LCPDAT1
  FDAT_ACT = FP3
  BAS(#CP_PARAMS, 0.5)
  SET_CD_PARAMS (0)
  TRIGGER WHEN DISTANCE = 1 DELAY = ArcGetDelay(#PreDefinition, WDAT1) DO ArcMainNG(#PreDefinition, WDAT1, WP3) PRIO = -1
  TRIGGER WHEN PATH = ArcGetPath(#OnTheFlyArcOn, WDAT1) DELAY = ArcGetDelay(#GasPreflow, WDAT1) DO ArcMainNG(#GasPreflow, WDAT1, WP3) PRIO = -1
  TRIGGER WHEN PATH = ArcGetPath(#OnTheFlyArcOn, WDAT1) DELAY = 0 DO ArcMainNG(#ArcOnMoveStd, WDAT1, WP3) PRIO = -1
  ArcMainNG(#ArcOnBeforeMoveStd, WDAT1, WP3)
  LIN XP3
  ArcMainNG(#ArcOnAfterMoveStd, WDAT1, WP3)
;ENDFOLD
   $VEL.CP = 0.025
   LIN  {X 4.181, Y -8.829, Z 19.500, A 0.000, B 0.000, C 0.000} C_DIS
   $VEL.CP = 0.060
   LIN  {X 8.829, Y -4.181, Z 19.500, A 0.000, B 0.000, C 0.000} C_DIS

;FOLD ARCOFF WDAT2 LIN P4 CPDAT2 Tool[1]:cmttorch Base[1]:vrashatel ;%{PE}
  ;FOLD Parameters ;%{h}
    ;Params IlfProvider=kukaroboter.arctech.arcofflin; Kuka.IsGlobalPoint=False; Kuka.PointName=P4; Kuka.BlendingEnabled=False; Kuka.MoveDataName=CPDAT2; Kuka.VelocityPath=0.01; Kuka.CurrentCDSetIndex=0; Kuka.MovementParameterFieldEnabled=True; ArcTech.WdatVarName=WDAT2; ArcTech.Basic=3.4.3.1264
  ;ENDFOLD
  $BWDSTART = FALSE
  LDAT_ACT = LCPDAT2
  FDAT_ACT = FP4
  BAS(#CP_PARAMS, gArcBasVelDefinition)
  SET_CD_PARAMS (0)
  TRIGGER WHEN PATH = ArcGetPath(#ArcOffBefore, WDAT2) DELAY = 0 DO ArcMainNG(#ArcOffBeforeOffStd, WDAT2, WP4) PRIO = -1
  TRIGGER WHEN PATH = ArcGetPath(#OnTheFlyArcOff, WDAT2) DELAY = 0 DO ArcMainNG(#ArcOffMoveStd, WDAT2, WP4) PRIO = -1
  ArcMainNG(#ArcOffBeforeMoveStd, WDAT2, WP4)
  LIN XP4
  ArcMainNG(#ArcOffAfterMoveStd, WDAT2, WP4)
;ENDFOLD
   $VEL.CP = 0.080
   LIN  {X 8.829, Y -4.746, Z 19.500, A 0.000, B 0.000, C 0.000} C_DIS

;FOLD ARCON WDAT1 LIN P3 Vel=0.5 m/s CPDAT1 Tool[1]:cmttorch Base[1]:vrashatel ;%{PE}
  ;FOLD Parameters ;%{h}
    ;Params IlfProvider=kukaroboter.arctech.arconlin; Kuka.IsGlobalPoint=False; Kuka.PointName=P3; Kuka.BlendingEnabled=False; Kuka.MoveDataName=CPDAT1; Kuka.VelocityPath=0.5; Kuka.CurrentCDSetIndex=0; Kuka.MovementParameterFieldEnabled=True; ArcTech.WdatVarName=WDAT1; ArcTech.Basic=3.4.3.1264
  ;ENDFOLD
  $BWDSTART = FALSE
  LDAT_ACT = LCPDAT1
  FDAT_ACT = FP3
  BAS(#CP_PARAMS, 0.5)
  SET_CD_PARAMS (0)
  TRIGGER WHEN DISTANCE = 1 DELAY = ArcGetDelay(#PreDefinition, WDAT1) DO ArcMainNG(#PreDefinition, WDAT1, WP3) PRIO = -1
  TRIGGER WHEN PATH = ArcGetPath(#OnTheFlyArcOn, WDAT1) DELAY = ArcGetDelay(#GasPreflow, WDAT1) DO ArcMainNG(#GasPreflow, WDAT1, WP3) PRIO = -1
  TRIGGER WHEN PATH = ArcGetPath(#OnTheFlyArcOn, WDAT1) DELAY = 0 DO ArcMainNG(#ArcOnMoveStd, WDAT1, WP3) PRIO = -1
  ArcMainNG(#ArcOnBeforeMoveStd, WDAT1, WP3)
  LIN XP3
  ArcMainNG(#ArcOnAfterMoveStd, WDAT1, WP3)
;ENDFOLD
   $VEL.CP = 0.060
   LIN  {X 4.746, Y -8.829, Z 19.500, A 0.000, B 0.000, C 0.000} C_DIS

;FOLD ARCOFF WDAT2 LIN P4 CPDAT2 Tool[1]:cmttorch Base[1]:vrashatel ;%{PE}
  ;FOLD Parameters ;%{h}
    ;Params IlfProvider=kukaroboter.arctech.arcofflin; Kuka.IsGlobalPoint=False; Kuka.PointName=P4; Kuka.BlendingEnabled=False; Kuka.MoveDataName=CPDAT2; Kuka.VelocityPath=0.01; Kuka.CurrentCDSetIndex=0; Kuka.MovementParameterFieldEnabled=True; ArcTech.WdatVarName=WDAT2; ArcTech.Basic=3.4.3.1264
  ;ENDFOLD
  $BWDSTART = FALSE
  LDAT_ACT = LCPDAT2
  FDAT_ACT = FP4
  BAS(#CP_PARAMS, gArcBasVelDefinition)
  SET_CD_PARAMS (0)
  TRIGGER WHEN PATH = ArcGetPath(#ArcOffBefore, WDAT2) DELAY = 0 DO ArcMainNG(#ArcOffBeforeOffStd, WDAT2, WP4) PRIO = -1
  TRIGGER WHEN PATH = ArcGetPath(#OnTheFlyArcOff, WDAT2) DELAY = 0 DO ArcMainNG(#ArcOffMoveStd, WDAT2, WP4) PRIO = -1
  ArcMainNG(#ArcOffBeforeMoveStd, WDAT2, WP4)
  LIN XP4
  ArcMainNG(#ArcOffAfterMoveStd, WDAT2, WP4)
;ENDFOLD
   $VEL.CP = 0.080
   LIN  {X 5.312, Y -8.829, Z 19.500, A 0.000, B 0.000, C 0.000} C_DIS

;FOLD ARCON WDAT1 LIN P3 Vel=0.5 m/s CPDAT1 Tool[1]:cmttorch Base[1]:vrashatel ;%{PE}
  ;FOLD Parameters ;%{h}
    ;Params IlfProvider=kukaroboter.arctech.arconlin; Kuka.IsGlobalPoint=False; Kuka.PointName=P3; Kuka.BlendingEnabled=False; Kuka.MoveDataName=CPDAT1; Kuka.VelocityPath=0.5; Kuka.CurrentCDSetIndex=0; Kuka.MovementParameterFieldEnabled=True; ArcTech.WdatVarName=WDAT1; ArcTech.Basic=3.4.3.1264
  ;ENDFOLD
  $BWDSTART = FALSE
  LDAT_ACT = LCPDAT1
  FDAT_ACT = FP3
  BAS(#CP_PARAMS, 0.5)
  SET_CD_PARAMS (0)
  TRIGGER WHEN DISTANCE = 1 DELAY = ArcGetDelay(#PreDefinition, WDAT1) DO ArcMainNG(#PreDefinition, WDAT1, WP3) PRIO = -1
  TRIGGER WHEN PATH = ArcGetPath(#OnTheFlyArcOn, WDAT1) DELAY = ArcGetDelay(#GasPreflow, WDAT1) DO ArcMainNG(#GasPreflow, WDAT1, WP3) PRIO = -1
  TRIGGER WHEN PATH = ArcGetPath(#OnTheFlyArcOn, WDAT1) DELAY = 0 DO ArcMainNG(#ArcOnMoveStd, WDAT1, WP3) PRIO = -1
  ArcMainNG(#ArcOnBeforeMoveStd, WDAT1, WP3)
  LIN XP3
  ArcMainNG(#ArcOnAfterMoveStd, WDAT1, WP3)
;ENDFOLD
   $VEL.CP = 0.060
   LIN  {X 8.829, Y -5.312, Z 19.500, A 0.000, B 0.000, C 0.000} C_DIS

;FOLD ARCOFF WDAT2 LIN P4 CPDAT2 Tool[1]:cmttorch Base[1]:vrashatel ;%{PE}
  ;FOLD Parameters ;%{h}
    ;Params IlfProvider=kukaroboter.arctech.arcofflin; Kuka.IsGlobalPoint=False; Kuka.PointName=P4; Kuka.BlendingEnabled=False; Kuka.MoveDataName=CPDAT2; Kuka.VelocityPath=0.01; Kuka.CurrentCDSetIndex=0; Kuka.MovementParameterFieldEnabled=True; ArcTech.WdatVarName=WDAT2; ArcTech.Basic=3.4.3.1264
  ;ENDFOLD
  $BWDSTART = FALSE
  LDAT_ACT = LCPDAT2
  FDAT_ACT = FP4
  BAS(#CP_PARAMS, gArcBasVelDefinition)
  SET_CD_PARAMS (0)
  TRIGGER WHEN PATH = ArcGetPath(#ArcOffBefore, WDAT2) DELAY = 0 DO ArcMainNG(#ArcOffBeforeOffStd, WDAT2, WP4) PRIO = -1
  TRIGGER WHEN PATH = ArcGetPath(#OnTheFlyArcOff, WDAT2) DELAY = 0 DO ArcMainNG(#ArcOffMoveStd, WDAT2, WP4) PRIO = -1
  ArcMainNG(#ArcOffBeforeMoveStd, WDAT2, WP4)
  LIN XP4
  ArcMainNG(#ArcOffAfterMoveStd, WDAT2, WP4)
;ENDFOLD
   $VEL.CP = 0.080
   LIN  {X 8.829, Y -5.878, Z 19.500, A 0.000, B 0.000, C 0.000} C_DIS

;FOLD ARCON WDAT1 LIN P3 Vel=0.5 m/s CPDAT1 Tool[1]:cmttorch Base[1]:vrashatel ;%{PE}
  ;FOLD Parameters ;%{h}
    ;Params IlfProvider=kukaroboter.arctech.arconlin; Kuka.IsGlobalPoint=False; Kuka.PointName=P3; Kuka.BlendingEnabled=False; Kuka.MoveDataName=CPDAT1; Kuka.VelocityPath=0.5; Kuka.CurrentCDSetIndex=0; Kuka.MovementParameterFieldEnabled=True; ArcTech.WdatVarName=WDAT1; ArcTech.Basic=3.4.3.1264
  ;ENDFOLD
  $BWDSTART = FALSE
  LDAT_ACT = LCPDAT1
  FDAT_ACT = FP3
  BAS(#CP_PARAMS, 0.5)
  SET_CD_PARAMS (0)
  TRIGGER WHEN DISTANCE = 1 DELAY = ArcGetDelay(#PreDefinition, WDAT1) DO ArcMainNG(#PreDefinition, WDAT1, WP3) PRIO = -1
  TRIGGER WHEN PATH = ArcGetPath(#OnTheFlyArcOn, WDAT1) DELAY = ArcGetDelay(#GasPreflow, WDAT1) DO ArcMainNG(#GasPreflow, WDAT1, WP3) PRIO = -1
  TRIGGER WHEN PATH = ArcGetPath(#OnTheFlyArcOn, WDAT1) DELAY = 0 DO ArcMainNG(#ArcOnMoveStd, WDAT1, WP3) PRIO = -1
  ArcMainNG(#ArcOnBeforeMoveStd, WDAT1, WP3)
  LIN XP3
  ArcMainNG(#ArcOnAfterMoveStd, WDAT1, WP3)
;ENDFOLD
   $VEL.CP = 0.060
   LIN  {X 5.878, Y -8.829, Z 19.500, A 0.000, B 0.000, C 0.000} C_DIS

;FOLD ARCOFF WDAT2 LIN P4 CPDAT2 Tool[1]:cmttorch Base[1]:vrashatel ;%{PE}
  ;FOLD Parameters ;%{h}
    ;Params IlfProvider=kukaroboter.arctech.arcofflin; Kuka.IsGlobalPoint=False; Kuka.PointName=P4; Kuka.BlendingEnabled=False; Kuka.MoveDataName=CPDAT2; Kuka.VelocityPath=0.01; Kuka.CurrentCDSetIndex=0; Kuka.MovementParameterFieldEnabled=True; ArcTech.WdatVarName=WDAT2; ArcTech.Basic=3.4.3.1264
  ;ENDFOLD
  $BWDSTART = FALSE
  LDAT_ACT = LCPDAT2
  FDAT_ACT = FP4
  BAS(#CP_PARAMS, gArcBasVelDefinition)
  SET_CD_PARAMS (0)
  TRIGGER WHEN PATH = ArcGetPath(#ArcOffBefore, WDAT2) DELAY = 0 DO ArcMainNG(#ArcOffBeforeOffStd, WDAT2, WP4) PRIO = -1
  TRIGGER WHEN PATH = ArcGetPath(#OnTheFlyArcOff, WDAT2) DELAY = 0 DO ArcMainNG(#ArcOffMoveStd, WDAT2, WP4) PRIO = -1
  ArcMainNG(#ArcOffBeforeMoveStd, WDAT2, WP4)
  LIN XP4
  ArcMainNG(#ArcOffAfterMoveStd, WDAT2, WP4)
;ENDFOLD
   $VEL.CP = 0.080
   LIN  {X 6.443, Y -8.829, Z 19.500, A 0.000, B 0.000, C 0.000} C_DIS

;FOLD ARCON WDAT1 LIN P3 Vel=0.5 m/s CPDAT1 Tool[1]:cmttorch Base[1]:vrashatel ;%{PE}
  ;FOLD Parameters ;%{h}
    ;Params IlfProvider=kukaroboter.arctech.arconlin; Kuka.IsGlobalPoint=False; Kuka.PointName=P3; Kuka.BlendingEnabled=False; Kuka.MoveDataName=CPDAT1; Kuka.VelocityPath=0.5; Kuka.CurrentCDSetIndex=0; Kuka.MovementParameterFieldEnabled=True; ArcTech.WdatVarName=WDAT1; ArcTech.Basic=3.4.3.1264
  ;ENDFOLD
  $BWDSTART = FALSE
  LDAT_ACT = LCPDAT1
  FDAT_ACT = FP3
  BAS(#CP_PARAMS, 0.5)
  SET_CD_PARAMS (0)
  TRIGGER WHEN DISTANCE = 1 DELAY = ArcGetDelay(#PreDefinition, WDAT1) DO ArcMainNG(#PreDefinition, WDAT1, WP3) PRIO = -1
  TRIGGER WHEN PATH = ArcGetPath(#OnTheFlyArcOn, WDAT1) DELAY = ArcGetDelay(#GasPreflow, WDAT1) DO ArcMainNG(#GasPreflow, WDAT1, WP3) PRIO = -1
  TRIGGER WHEN PATH = ArcGetPath(#OnTheFlyArcOn, WDAT1) DELAY = 0 DO ArcMainNG(#ArcOnMoveStd, WDAT1, WP3) PRIO = -1
  ArcMainNG(#ArcOnBeforeMoveStd, WDAT1, WP3)
  LIN XP3
  ArcMainNG(#ArcOnAfterMoveStd, WDAT1, WP3)
;ENDFOLD
   $VEL.CP = 0.060
   LIN  {X 8.829, Y -6.443, Z 19.500, A 0.000, B 0.000, C 0.000} C_DIS

;FOLD ARCOFF WDAT2 LIN P4 CPDAT2 Tool[1]:cmttorch Base[1]:vrashatel ;%{PE}
  ;FOLD Parameters ;%{h}
    ;Params IlfProvider=kukaroboter.arctech.arcofflin; Kuka.IsGlobalPoint=False; Kuka.PointName=P4; Kuka.BlendingEnabled=False; Kuka.MoveDataName=CPDAT2; Kuka.VelocityPath=0.01; Kuka.CurrentCDSetIndex=0; Kuka.MovementParameterFieldEnabled=True; ArcTech.WdatVarName=WDAT2; ArcTech.Basic=3.4.3.1264
  ;ENDFOLD
  $BWDSTART = FALSE
  LDAT_ACT = LCPDAT2
  FDAT_ACT = FP4
  BAS(#CP_PARAMS, gArcBasVelDefinition)
  SET_CD_PARAMS (0)
  TRIGGER WHEN PATH = ArcGetPath(#ArcOffBefore, WDAT2) DELAY = 0 DO ArcMainNG(#ArcOffBeforeOffStd, WDAT2, WP4) PRIO = -1
  TRIGGER WHEN PATH = ArcGetPath(#OnTheFlyArcOff, WDAT2) DELAY = 0 DO ArcMainNG(#ArcOffMoveStd, WDAT2, WP4) PRIO = -1
  ArcMainNG(#ArcOffBeforeMoveStd, WDAT2, WP4)
  LIN XP4
  ArcMainNG(#ArcOffAfterMoveStd, WDAT2, WP4)
;ENDFOLD
   $VEL.CP = 0.080
   LIN  {X 8.829, Y -7.009, Z 19.500, A 0.000, B 0.000, C 0.000} C_DIS

;FOLD ARCON WDAT1 LIN P3 Vel=0.5 m/s CPDAT1 Tool[1]:cmttorch Base[1]:vrashatel ;%{PE}
  ;FOLD Parameters ;%{h}
    ;Params IlfProvider=kukaroboter.arctech.arconlin; Kuka.IsGlobalPoint=False; Kuka.PointName=P3; Kuka.BlendingEnabled=False; Kuka.MoveDataName=CPDAT1; Kuka.VelocityPath=0.5; Kuka.CurrentCDSetIndex=0; Kuka.MovementParameterFieldEnabled=True; ArcTech.WdatVarName=WDAT1; ArcTech.Basic=3.4.3.1264
  ;ENDFOLD
  $BWDSTART = FALSE
  LDAT_ACT = LCPDAT1
  FDAT_ACT = FP3
  BAS(#CP_PARAMS, 0.5)
  SET_CD_PARAMS (0)
  TRIGGER WHEN DISTANCE = 1 DELAY = ArcGetDelay(#PreDefinition, WDAT1) DO ArcMainNG(#PreDefinition, WDAT1, WP3) PRIO = -1
  TRIGGER WHEN PATH = ArcGetPath(#OnTheFlyArcOn, WDAT1) DELAY = ArcGetDelay(#GasPreflow, WDAT1) DO ArcMainNG(#GasPreflow, WDAT1, WP3) PRIO = -1
  TRIGGER WHEN PATH = ArcGetPath(#OnTheFlyArcOn, WDAT1) DELAY = 0 DO ArcMainNG(#ArcOnMoveStd, WDAT1, WP3) PRIO = -1
  ArcMainNG(#ArcOnBeforeMoveStd, WDAT1, WP3)
  LIN XP3
  ArcMainNG(#ArcOnAfterMoveStd, WDAT1, WP3)
;ENDFOLD
   $VEL.CP = 0.060
   LIN  {X 7.009, Y -8.829, Z 19.500, A 0.000, B 0.000, C 0.000} C_DIS

;FOLD ARCOFF WDAT2 LIN P4 CPDAT2 Tool[1]:cmttorch Base[1]:vrashatel ;%{PE}
  ;FOLD Parameters ;%{h}
    ;Params IlfProvider=kukaroboter.arctech.arcofflin; Kuka.IsGlobalPoint=False; Kuka.PointName=P4; Kuka.BlendingEnabled=False; Kuka.MoveDataName=CPDAT2; Kuka.VelocityPath=0.01; Kuka.CurrentCDSetIndex=0; Kuka.MovementParameterFieldEnabled=True; ArcTech.WdatVarName=WDAT2; ArcTech.Basic=3.4.3.1264
  ;ENDFOLD
  $BWDSTART = FALSE
  LDAT_ACT = LCPDAT2
  FDAT_ACT = FP4
  BAS(#CP_PARAMS, gArcBasVelDefinition)
  SET_CD_PARAMS (0)
  TRIGGER WHEN PATH = ArcGetPath(#ArcOffBefore, WDAT2) DELAY = 0 DO ArcMainNG(#ArcOffBeforeOffStd, WDAT2, WP4) PRIO = -1
  TRIGGER WHEN PATH = ArcGetPath(#OnTheFlyArcOff, WDAT2) DELAY = 0 DO ArcMainNG(#ArcOffMoveStd, WDAT2, WP4) PRIO = -1
  ArcMainNG(#ArcOffBeforeMoveStd, WDAT2, WP4)
  LIN XP4
  ArcMainNG(#ArcOffAfterMoveStd, WDAT2, WP4)
;ENDFOLD
   $VEL.CP = 0.080
   LIN  {X 7.575, Y -8.829, Z 19.500, A 0.000, B 0.000, C 0.000} C_DIS

;FOLD ARCON WDAT1 LIN P3 Vel=0.5 m/s CPDAT1 Tool[1]:cmttorch Base[1]:vrashatel ;%{PE}
  ;FOLD Parameters ;%{h}
    ;Params IlfProvider=kukaroboter.arctech.arconlin; Kuka.IsGlobalPoint=False; Kuka.PointName=P3; Kuka.BlendingEnabled=False; Kuka.MoveDataName=CPDAT1; Kuka.VelocityPath=0.5; Kuka.CurrentCDSetIndex=0; Kuka.MovementParameterFieldEnabled=True; ArcTech.WdatVarName=WDAT1; ArcTech.Basic=3.4.3.1264
  ;ENDFOLD
  $BWDSTART = FALSE
  LDAT_ACT = LCPDAT1
  FDAT_ACT = FP3
  BAS(#CP_PARAMS, 0.5)
  SET_CD_PARAMS (0)
  TRIGGER WHEN DISTANCE = 1 DELAY = ArcGetDelay(#PreDefinition, WDAT1) DO ArcMainNG(#PreDefinition, WDAT1, WP3) PRIO = -1
  TRIGGER WHEN PATH = ArcGetPath(#OnTheFlyArcOn, WDAT1) DELAY = ArcGetDelay(#GasPreflow, WDAT1) DO ArcMainNG(#GasPreflow, WDAT1, WP3) PRIO = -1
  TRIGGER WHEN PATH = ArcGetPath(#OnTheFlyArcOn, WDAT1) DELAY = 0 DO ArcMainNG(#ArcOnMoveStd, WDAT1, WP3) PRIO = -1
  ArcMainNG(#ArcOnBeforeMoveStd, WDAT1, WP3)
  LIN XP3
  ArcMainNG(#ArcOnAfterMoveStd, WDAT1, WP3)
;ENDFOLD
   $VEL.CP = 0.060
   LIN  {X 8.829, Y -7.575, Z 19.500, A 0.000, B 0.000, C 0.000} C_DIS

;FOLD ARCOFF WDAT2 LIN P4 CPDAT2 Tool[1]:cmttorch Base[1]:vrashatel ;%{PE}
  ;FOLD Parameters ;%{h}
    ;Params IlfProvider=kukaroboter.arctech.arcofflin; Kuka.IsGlobalPoint=False; Kuka.PointName=P4; Kuka.BlendingEnabled=False; Kuka.MoveDataName=CPDAT2; Kuka.VelocityPath=0.01; Kuka.CurrentCDSetIndex=0; Kuka.MovementParameterFieldEnabled=True; ArcTech.WdatVarName=WDAT2; ArcTech.Basic=3.4.3.1264
  ;ENDFOLD
  $BWDSTART = FALSE
  LDAT_ACT = LCPDAT2
  FDAT_ACT = FP4
  BAS(#CP_PARAMS, gArcBasVelDefinition)
  SET_CD_PARAMS (0)
  TRIGGER WHEN PATH = ArcGetPath(#ArcOffBefore, WDAT2) DELAY = 0 DO ArcMainNG(#ArcOffBeforeOffStd, WDAT2, WP4) PRIO = -1
  TRIGGER WHEN PATH = ArcGetPath(#OnTheFlyArcOff, WDAT2) DELAY = 0 DO ArcMainNG(#ArcOffMoveStd, WDAT2, WP4) PRIO = -1
  ArcMainNG(#ArcOffBeforeMoveStd, WDAT2, WP4)
  LIN XP4
  ArcMainNG(#ArcOffAfterMoveStd, WDAT2, WP4)
;ENDFOLD
   $VEL.CP = 0.080
   LIN  {X 8.829, Y -8.140, Z 19.500, A 0.000, B 0.000, C 0.000} C_DIS

;FOLD ARCON WDAT1 LIN P3 Vel=0.5 m/s CPDAT1 Tool[1]:cmttorch Base[1]:vrashatel ;%{PE}
  ;FOLD Parameters ;%{h}
    ;Params IlfProvider=kukaroboter.arctech.arconlin; Kuka.IsGlobalPoint=False; Kuka.PointName=P3; Kuka.BlendingEnabled=False; Kuka.MoveDataName=CPDAT1; Kuka.VelocityPath=0.5; Kuka.CurrentCDSetIndex=0; Kuka.MovementParameterFieldEnabled=True; ArcTech.WdatVarName=WDAT1; ArcTech.Basic=3.4.3.1264
  ;ENDFOLD
  $BWDSTART = FALSE
  LDAT_ACT = LCPDAT1
  FDAT_ACT = FP3
  BAS(#CP_PARAMS, 0.5)
  SET_CD_PARAMS (0)
  TRIGGER WHEN DISTANCE = 1 DELAY = ArcGetDelay(#PreDefinition, WDAT1) DO ArcMainNG(#PreDefinition, WDAT1, WP3) PRIO = -1
  TRIGGER WHEN PATH = ArcGetPath(#OnTheFlyArcOn, WDAT1) DELAY = ArcGetDelay(#GasPreflow, WDAT1) DO ArcMainNG(#GasPreflow, WDAT1, WP3) PRIO = -1
  TRIGGER WHEN PATH = ArcGetPath(#OnTheFlyArcOn, WDAT1) DELAY = 0 DO ArcMainNG(#ArcOnMoveStd, WDAT1, WP3) PRIO = -1
  ArcMainNG(#ArcOnBeforeMoveStd, WDAT1, WP3)
  LIN XP3
  ArcMainNG(#ArcOnAfterMoveStd, WDAT1, WP3)
;ENDFOLD
   $VEL.CP = 0.060
   LIN  {X 8.140, Y -8.829, Z 19.500, A 0.000, B 0.000, C 0.000} C_DIS

;FOLD ARCOFF WDAT2 LIN P4 CPDAT2 Tool[1]:cmttorch Base[1]:vrashatel ;%{PE}
  ;FOLD Parameters ;%{h}
    ;Params IlfProvider=kukaroboter.arctech.arcofflin; Kuka.IsGlobalPoint=False; Kuka.PointName=P4; Kuka.BlendingEnabled=False; Kuka.MoveDataName=CPDAT2; Kuka.VelocityPath=0.01; Kuka.CurrentCDSetIndex=0; Kuka.MovementParameterFieldEnabled=True; ArcTech.WdatVarName=WDAT2; ArcTech.Basic=3.4.3.1264
  ;ENDFOLD
  $BWDSTART = FALSE
  LDAT_ACT = LCPDAT2
  FDAT_ACT = FP4
  BAS(#CP_PARAMS, gArcBasVelDefinition)
  SET_CD_PARAMS (0)
  TRIGGER WHEN PATH = ArcGetPath(#ArcOffBefore, WDAT2) DELAY = 0 DO ArcMainNG(#ArcOffBeforeOffStd, WDAT2, WP4) PRIO = -1
  TRIGGER WHEN PATH = ArcGetPath(#OnTheFlyArcOff, WDAT2) DELAY = 0 DO ArcMainNG(#ArcOffMoveStd, WDAT2, WP4) PRIO = -1
  ArcMainNG(#ArcOffBeforeMoveStd, WDAT2, WP4)
  LIN XP4
  ArcMainNG(#ArcOffAfterMoveStd, WDAT2, WP4)
;ENDFOLD
   $VEL.CP = 0.080
   LIN  {X 8.706, Y -8.829, Z 19.500, A 0.000, B 0.000, C 0.000} C_DIS

;FOLD ARCON WDAT1 LIN P3 Vel=0.5 m/s CPDAT1 Tool[1]:cmttorch Base[1]:vrashatel ;%{PE}
  ;FOLD Parameters ;%{h}
    ;Params IlfProvider=kukaroboter.arctech.arconlin; Kuka.IsGlobalPoint=False; Kuka.PointName=P3; Kuka.BlendingEnabled=False; Kuka.MoveDataName=CPDAT1; Kuka.VelocityPath=0.5; Kuka.CurrentCDSetIndex=0; Kuka.MovementParameterFieldEnabled=True; ArcTech.WdatVarName=WDAT1; ArcTech.Basic=3.4.3.1264
  ;ENDFOLD
  $BWDSTART = FALSE
  LDAT_ACT = LCPDAT1
  FDAT_ACT = FP3
  BAS(#CP_PARAMS, 0.5)
  SET_CD_PARAMS (0)
  TRIGGER WHEN DISTANCE = 1 DELAY = ArcGetDelay(#PreDefinition, WDAT1) DO ArcMainNG(#PreDefinition, WDAT1, WP3) PRIO = -1
  TRIGGER WHEN PATH = ArcGetPath(#OnTheFlyArcOn, WDAT1) DELAY = ArcGetDelay(#GasPreflow, WDAT1) DO ArcMainNG(#GasPreflow, WDAT1, WP3) PRIO = -1
  TRIGGER WHEN PATH = ArcGetPath(#OnTheFlyArcOn, WDAT1) DELAY = 0 DO ArcMainNG(#ArcOnMoveStd, WDAT1, WP3) PRIO = -1
  ArcMainNG(#ArcOnBeforeMoveStd, WDAT1, WP3)
  LIN XP3
  ArcMainNG(#ArcOnAfterMoveStd, WDAT1, WP3)
;ENDFOLD
   $VEL.CP = 0.060
   LIN  {X 8.829, Y -8.706, Z 19.500, A 0.000, B 0.000, C 0.000} C_DIS

;FOLD ARCOFF WDAT2 LIN P4 CPDAT2 Tool[1]:cmttorch Base[1]:vrashatel ;%{PE}
  ;FOLD Parameters ;%{h}
    ;Params IlfProvider=kukaroboter.arctech.arcofflin; Kuka.IsGlobalPoint=False; Kuka.PointName=P4; Kuka.BlendingEnabled=False; Kuka.MoveDataName=CPDAT2; Kuka.VelocityPath=0.01; Kuka.CurrentCDSetIndex=0; Kuka.MovementParameterFieldEnabled=True; ArcTech.WdatVarName=WDAT2; ArcTech.Basic=3.4.3.1264
  ;ENDFOLD
  $BWDSTART = FALSE
  LDAT_ACT = LCPDAT2
  FDAT_ACT = FP4
  BAS(#CP_PARAMS, gArcBasVelDefinition)
  SET_CD_PARAMS (0)
  TRIGGER WHEN PATH = ArcGetPath(#ArcOffBefore, WDAT2) DELAY = 0 DO ArcMainNG(#ArcOffBeforeOffStd, WDAT2, WP4) PRIO = -1
  TRIGGER WHEN PATH = ArcGetPath(#OnTheFlyArcOff, WDAT2) DELAY = 0 DO ArcMainNG(#ArcOffMoveStd, WDAT2, WP4) PRIO = -1
  ArcMainNG(#ArcOffBeforeMoveStd, WDAT2, WP4)
  LIN XP4
  ArcMainNG(#ArcOffAfterMoveStd, WDAT2, WP4)
;ENDFOLD
   $VEL.CP = 0.080
   LIN  {X 9.200, Y -8.706, Z 19.500, A 0.000, B 0.000, C 0.000} C_DIS
   $VEL.CP = 0.010
   LIN  {X 9.200, Y -8.706, Z 19.700, A 0.000, B 0.000, C 0.000} C_DIS
   $VEL.CP = 0.080
   LIN  {X 9.290, Y -8.706, Z 19.700, A 0.000, B 0.000, C 0.000} C_DIS
   $VEL.CP = 0.080
   LIN  {X 9.218, Y 9.218, Z 19.700, A 0.000, B 0.000, C 0.000} C_DIS
   $VEL.CP = 0.080
   LIN  {X -9.530, Y 9.530, Z 19.700, A 0.000, B 0.000, C 0.000} C_DIS
   $VEL.CP = 0.080
   LIN  {X -9.800, Y 9.800, Z 19.700, A 0.000, B 0.000, C 0.000} C_DIS

;FOLD ARCON WDAT1 LIN P3 Vel=0.5 m/s CPDAT1 Tool[1]:cmttorch Base[1]:vrashatel ;%{PE}
  ;FOLD Parameters ;%{h}
    ;Params IlfProvider=kukaroboter.arctech.arconlin; Kuka.IsGlobalPoint=False; Kuka.PointName=P3; Kuka.BlendingEnabled=False; Kuka.MoveDataName=CPDAT1; Kuka.VelocityPath=0.5; Kuka.CurrentCDSetIndex=0; Kuka.MovementParameterFieldEnabled=True; ArcTech.WdatVarName=WDAT1; ArcTech.Basic=3.4.3.1264
  ;ENDFOLD
  $BWDSTART = FALSE
  LDAT_ACT = LCPDAT1
  FDAT_ACT = FP3
  BAS(#CP_PARAMS, 0.5)
  SET_CD_PARAMS (0)
  TRIGGER WHEN DISTANCE = 1 DELAY = ArcGetDelay(#PreDefinition, WDAT1) DO ArcMainNG(#PreDefinition, WDAT1, WP3) PRIO = -1
  TRIGGER WHEN PATH = ArcGetPath(#OnTheFlyArcOn, WDAT1) DELAY = ArcGetDelay(#GasPreflow, WDAT1) DO ArcMainNG(#GasPreflow, WDAT1, WP3) PRIO = -1
  TRIGGER WHEN PATH = ArcGetPath(#OnTheFlyArcOn, WDAT1) DELAY = 0 DO ArcMainNG(#ArcOnMoveStd, WDAT1, WP3) PRIO = -1
  ArcMainNG(#ArcOnBeforeMoveStd, WDAT1, WP3)
  LIN XP3
  ArcMainNG(#ArcOnAfterMoveStd, WDAT1, WP3)
;ENDFOLD
   $VEL.CP = 0.025
   LIN  {X -9.800, Y 9.800, Z 19.700, A 0.000, B 0.000, C 0.000} C_DIS
   $VEL.CP = 0.060
   LIN  {X -9.800, Y -9.800, Z 19.700, A 0.000, B 0.000, C 0.000} C_DIS
   $VEL.CP = 0.060
   LIN  {X 9.800, Y -9.800, Z 19.700, A 0.000, B 0.000, C 0.000} C_DIS
   $VEL.CP = 0.060
   LIN  {X 9.800, Y 9.800, Z 19.700, A 0.000, B 0.000, C 0.000} C_DIS
   $VEL.CP = 0.060
   LIN  {X -9.800, Y 9.800, Z 19.700, A 0.000, B 0.000, C 0.000} C_DIS

;FOLD ARCOFF WDAT2 LIN P4 CPDAT2 Tool[1]:cmttorch Base[1]:vrashatel ;%{PE}
  ;FOLD Parameters ;%{h}
    ;Params IlfProvider=kukaroboter.arctech.arcofflin; Kuka.IsGlobalPoint=False; Kuka.PointName=P4; Kuka.BlendingEnabled=False; Kuka.MoveDataName=CPDAT2; Kuka.VelocityPath=0.01; Kuka.CurrentCDSetIndex=0; Kuka.MovementParameterFieldEnabled=True; ArcTech.WdatVarName=WDAT2; ArcTech.Basic=3.4.3.1264
  ;ENDFOLD
  $BWDSTART = FALSE
  LDAT_ACT = LCPDAT2
  FDAT_ACT = FP4
  BAS(#CP_PARAMS, gArcBasVelDefinition)
  SET_CD_PARAMS (0)
  TRIGGER WHEN PATH = ArcGetPath(#ArcOffBefore, WDAT2) DELAY = 0 DO ArcMainNG(#ArcOffBeforeOffStd, WDAT2, WP4) PRIO = -1
  TRIGGER WHEN PATH = ArcGetPath(#OnTheFlyArcOff, WDAT2) DELAY = 0 DO ArcMainNG(#ArcOffMoveStd, WDAT2, WP4) PRIO = -1
  ArcMainNG(#ArcOffBeforeMoveStd, WDAT2, WP4)
  LIN XP4
  ArcMainNG(#ArcOffAfterMoveStd, WDAT2, WP4)
;ENDFOLD
   $VEL.CP = 0.080
   LIN  {X -9.800, Y 9.600, Z 19.700, A 0.000, B 0.000, C 0.000} C_DIS
   $VEL.CP = 0.080
   LIN  {X -9.360, Y 9.360, Z 19.700, A 0.000, B 0.000, C 0.000} C_DIS
   $VEL.CP = 0.080
   LIN  {X -4.094, Y 9.190, Z 19.700, A 0.000, B 0.000, C 0.000} C_DIS
   $VEL.CP = 0.080
   LIN  {X -4.094, Y 7.108, Z 19.700, A 0.000, B 0.000, C 0.000} C_DIS
   $VEL.CP = 0.080
   LIN  {X -4.094, Y 4.605, Z 19.700, A 0.000, B 0.000, C 0.000} C_DIS
   $VEL.CP = 0.080
   LIN  {X -3.794, Y 4.605, Z 19.700, A 0.000, B 0.000, C 0.000} C_DIS

;FOLD ARCON WDAT1 LIN P3 Vel=0.5 m/s CPDAT1 Tool[1]:cmttorch Base[1]:vrashatel ;%{PE}
  ;FOLD Parameters ;%{h}
    ;Params IlfProvider=kukaroboter.arctech.arconlin; Kuka.IsGlobalPoint=False; Kuka.PointName=P3; Kuka.BlendingEnabled=False; Kuka.MoveDataName=CPDAT1; Kuka.VelocityPath=0.5; Kuka.CurrentCDSetIndex=0; Kuka.MovementParameterFieldEnabled=True; ArcTech.WdatVarName=WDAT1; ArcTech.Basic=3.4.3.1264
  ;ENDFOLD
  $BWDSTART = FALSE
  LDAT_ACT = LCPDAT1
  FDAT_ACT = FP3
  BAS(#CP_PARAMS, 0.5)
  SET_CD_PARAMS (0)
  TRIGGER WHEN DISTANCE = 1 DELAY = ArcGetDelay(#PreDefinition, WDAT1) DO ArcMainNG(#PreDefinition, WDAT1, WP3) PRIO = -1
  TRIGGER WHEN PATH = ArcGetPath(#OnTheFlyArcOn, WDAT1) DELAY = ArcGetDelay(#GasPreflow, WDAT1) DO ArcMainNG(#GasPreflow, WDAT1, WP3) PRIO = -1
  TRIGGER WHEN PATH = ArcGetPath(#OnTheFlyArcOn, WDAT1) DELAY = 0 DO ArcMainNG(#ArcOnMoveStd, WDAT1, WP3) PRIO = -1
  ArcMainNG(#ArcOnBeforeMoveStd, WDAT1, WP3)
  LIN XP3
  ArcMainNG(#ArcOnAfterMoveStd, WDAT1, WP3)
;ENDFOLD
   $VEL.CP = 0.025
   LIN  {X -3.794, Y 4.605, Z 19.700, A 0.000, B 0.000, C 0.000} C_DIS
   $VEL.CP = 0.060
   LIN  {X -3.794, Y 6.518, Z 19.700, A 0.000, B 0.000, C 0.000} C_DIS
   $VEL.CP = 0.060
   LIN  {X 4.127, Y 6.518, Z 19.700, A 0.000, B 0.000, C 0.000} C_DIS
   $VEL.CP = 0.060
   LIN  {X 4.127, Y 5.850, Z 19.700, A 0.000, B 0.000, C 0.000} C_DIS
   $VEL.CP = 0.060
   LIN  {X -1.057, Y -4.280, Z 19.700, A 0.000, B 0.000, C 0.000} C_DIS
   $VEL.CP = 0.060
   LIN  {X 4.312, Y -4.280, Z 19.700, A 0.000, B 0.000, C 0.000} C_DIS
   $VEL.CP = 0.060
   LIN  {X 4.312, Y -6.193, Z 19.700, A 0.000, B 0.000, C 0.000} C_DIS
   $VEL.CP = 0.060
   LIN  {X -3.878, Y -6.193, Z 19.700, A 0.000, B 0.000, C 0.000} C_DIS
   $VEL.CP = 0.060
   LIN  {X -3.878, Y -5.525, Z 19.700, A 0.000, B 0.000, C 0.000} C_DIS
   $VEL.CP = 0.060
   LIN  {X 1.290, Y 4.605, Z 19.700, A 0.000, B 0.000, C 0.000} C_DIS
   $VEL.CP = 0.060
   LIN  {X -3.794, Y 4.605, Z 19.700, A 0.000, B 0.000, C 0.000} C_DIS

;FOLD ARCOFF WDAT2 LIN P4 CPDAT2 Tool[1]:cmttorch Base[1]:vrashatel ;%{PE}
  ;FOLD Parameters ;%{h}
    ;Params IlfProvider=kukaroboter.arctech.arcofflin; Kuka.IsGlobalPoint=False; Kuka.PointName=P4; Kuka.BlendingEnabled=False; Kuka.MoveDataName=CPDAT2; Kuka.VelocityPath=0.01; Kuka.CurrentCDSetIndex=0; Kuka.MovementParameterFieldEnabled=True; ArcTech.WdatVarName=WDAT2; ArcTech.Basic=3.4.3.1264
  ;ENDFOLD
  $BWDSTART = FALSE
  LDAT_ACT = LCPDAT2
  FDAT_ACT = FP4
  BAS(#CP_PARAMS, gArcBasVelDefinition)
  SET_CD_PARAMS (0)
  TRIGGER WHEN PATH = ArcGetPath(#ArcOffBefore, WDAT2) DELAY = 0 DO ArcMainNG(#ArcOffBeforeOffStd, WDAT2, WP4) PRIO = -1
  TRIGGER WHEN PATH = ArcGetPath(#OnTheFlyArcOff, WDAT2) DELAY = 0 DO ArcMainNG(#ArcOffMoveStd, WDAT2, WP4) PRIO = -1
  ArcMainNG(#ArcOffBeforeMoveStd, WDAT2, WP4)
  LIN XP4
  ArcMainNG(#ArcOffAfterMoveStd, WDAT2, WP4)
;ENDFOLD
   $VEL.CP = 0.080
   LIN  {X -3.794, Y 4.805, Z 19.700, A 0.000, B 0.000, C 0.000} C_DIS
   $VEL.CP = 0.080
   LIN  {X -4.194, Y 4.205, Z 19.700, A 0.000, B 0.000, C 0.000} C_DIS

;FOLD ARCON WDAT1 LIN P3 Vel=0.5 m/s CPDAT1 Tool[1]:cmttorch Base[1]:vrashatel ;%{PE}
  ;FOLD Parameters ;%{h}
    ;Params IlfProvider=kukaroboter.arctech.arconlin; Kuka.IsGlobalPoint=False; Kuka.PointName=P3; Kuka.BlendingEnabled=False; Kuka.MoveDataName=CPDAT1; Kuka.VelocityPath=0.5; Kuka.CurrentCDSetIndex=0; Kuka.MovementParameterFieldEnabled=True; ArcTech.WdatVarName=WDAT1; ArcTech.Basic=3.4.3.1264
  ;ENDFOLD
  $BWDSTART = FALSE
  LDAT_ACT = LCPDAT1
  FDAT_ACT = FP3
  BAS(#CP_PARAMS, 0.5)
  SET_CD_PARAMS (0)
  TRIGGER WHEN DISTANCE = 1 DELAY = ArcGetDelay(#PreDefinition, WDAT1) DO ArcMainNG(#PreDefinition, WDAT1, WP3) PRIO = -1
  TRIGGER WHEN PATH = ArcGetPath(#OnTheFlyArcOn, WDAT1) DELAY = ArcGetDelay(#GasPreflow, WDAT1) DO ArcMainNG(#GasPreflow, WDAT1, WP3) PRIO = -1
  TRIGGER WHEN PATH = ArcGetPath(#OnTheFlyArcOn, WDAT1) DELAY = 0 DO ArcMainNG(#ArcOnMoveStd, WDAT1, WP3) PRIO = -1
  ArcMainNG(#ArcOnBeforeMoveStd, WDAT1, WP3)
  LIN XP3
  ArcMainNG(#ArcOnAfterMoveStd, WDAT1, WP3)
;ENDFOLD
   $VEL.CP = 0.060
   LIN  {X -4.194, Y 6.918, Z 19.700, A 0.000, B 0.000, C 0.000} C_DIS
   $VEL.CP = 0.060
   LIN  {X 4.527, Y 6.918, Z 19.700, A 0.000, B 0.000, C 0.000} C_DIS
   $VEL.CP = 0.060
   LIN  {X 4.527, Y 5.754, Z 19.700, A 0.000, B 0.000, C 0.000} C_DIS
   $VEL.CP = 0.060
   LIN  {X -0.403, Y -3.880, Z 19.700, A 0.000, B 0.000, C 0.000} C_DIS
   $VEL.CP = 0.060
   LIN  {X 4.712, Y -3.880, Z 19.700, A 0.000, B 0.000, C 0.000} C_DIS
   $VEL.CP = 0.060
   LIN  {X 4.712, Y -6.593, Z 19.700, A 0.000, B 0.000, C 0.000} C_DIS
   $VEL.CP = 0.060
   LIN  {X -4.278, Y -6.593, Z 19.700, A 0.000, B 0.000, C 0.000} C_DIS
   $VEL.CP = 0.060
   LIN  {X -4.278, Y -5.429, Z 19.700, A 0.000, B 0.000, C 0.000} C_DIS
   $VEL.CP = 0.060
   LIN  {X 0.637, Y 4.205, Z 19.700, A 0.000, B 0.000, C 0.000} C_DIS
   $VEL.CP = 0.060
   LIN  {X -4.194, Y 4.205, Z 19.700, A 0.000, B 0.000, C 0.000} C_DIS

;FOLD ARCOFF WDAT2 LIN P4 CPDAT2 Tool[1]:cmttorch Base[1]:vrashatel ;%{PE}
  ;FOLD Parameters ;%{h}
    ;Params IlfProvider=kukaroboter.arctech.arcofflin; Kuka.IsGlobalPoint=False; Kuka.PointName=P4; Kuka.BlendingEnabled=False; Kuka.MoveDataName=CPDAT2; Kuka.VelocityPath=0.01; Kuka.CurrentCDSetIndex=0; Kuka.MovementParameterFieldEnabled=True; ArcTech.WdatVarName=WDAT2; ArcTech.Basic=3.4.3.1264
  ;ENDFOLD
  $BWDSTART = FALSE
  LDAT_ACT = LCPDAT2
  FDAT_ACT = FP4
  BAS(#CP_PARAMS, gArcBasVelDefinition)
  SET_CD_PARAMS (0)
  TRIGGER WHEN PATH = ArcGetPath(#ArcOffBefore, WDAT2) DELAY = 0 DO ArcMainNG(#ArcOffBeforeOffStd, WDAT2, WP4) PRIO = -1
  TRIGGER WHEN PATH = ArcGetPath(#OnTheFlyArcOff, WDAT2) DELAY = 0 DO ArcMainNG(#ArcOffMoveStd, WDAT2, WP4) PRIO = -1
  ArcMainNG(#ArcOffBeforeMoveStd, WDAT2, WP4)
  LIN XP4
  ArcMainNG(#ArcOffAfterMoveStd, WDAT2, WP4)
;ENDFOLD
   $VEL.CP = 0.080
   LIN  {X -4.390, Y 7.114, Z 19.700, A 0.000, B 0.000, C 0.000} C_DIS
   $VEL.CP = 0.080
   LIN  {X -4.390, Y 9.190, Z 19.700, A 0.000, B 0.000, C 0.000} C_DIS
   $VEL.CP = 0.080
   LIN  {X -9.400, Y 9.400, Z 19.700, A 0.000, B 0.000, C 0.000} C_DIS

;FOLD ARCON WDAT1 LIN P3 Vel=0.5 m/s CPDAT1 Tool[1]:cmttorch Base[1]:vrashatel ;%{PE}
  ;FOLD Parameters ;%{h}
    ;Params IlfProvider=kukaroboter.arctech.arconlin; Kuka.IsGlobalPoint=False; Kuka.PointName=P3; Kuka.BlendingEnabled=False; Kuka.MoveDataName=CPDAT1; Kuka.VelocityPath=0.5; Kuka.CurrentCDSetIndex=0; Kuka.MovementParameterFieldEnabled=True; ArcTech.WdatVarName=WDAT1; ArcTech.Basic=3.4.3.1264
  ;ENDFOLD
  $BWDSTART = FALSE
  LDAT_ACT = LCPDAT1
  FDAT_ACT = FP3
  BAS(#CP_PARAMS, 0.5)
  SET_CD_PARAMS (0)
  TRIGGER WHEN DISTANCE = 1 DELAY = ArcGetDelay(#PreDefinition, WDAT1) DO ArcMainNG(#PreDefinition, WDAT1, WP3) PRIO = -1
  TRIGGER WHEN PATH = ArcGetPath(#OnTheFlyArcOn, WDAT1) DELAY = ArcGetDelay(#GasPreflow, WDAT1) DO ArcMainNG(#GasPreflow, WDAT1, WP3) PRIO = -1
  TRIGGER WHEN PATH = ArcGetPath(#OnTheFlyArcOn, WDAT1) DELAY = 0 DO ArcMainNG(#ArcOnMoveStd, WDAT1, WP3) PRIO = -1
  ArcMainNG(#ArcOnBeforeMoveStd, WDAT1, WP3)
  LIN XP3
  ArcMainNG(#ArcOnAfterMoveStd, WDAT1, WP3)
;ENDFOLD
   $VEL.CP = 0.025
   LIN  {X -9.400, Y 9.400, Z 19.700, A 0.000, B 0.000, C 0.000} C_DIS
   $VEL.CP = 0.060
   LIN  {X -9.400, Y -9.400, Z 19.700, A 0.000, B 0.000, C 0.000} C_DIS
   $VEL.CP = 0.060
   LIN  {X 9.400, Y -9.400, Z 19.700, A 0.000, B 0.000, C 0.000} C_DIS
   $VEL.CP = 0.060
   LIN  {X 9.400, Y 9.400, Z 19.700, A 0.000, B 0.000, C 0.000} C_DIS
   $VEL.CP = 0.060
   LIN  {X -9.400, Y 9.400, Z 19.700, A 0.000, B 0.000, C 0.000} C_DIS

;FOLD ARCOFF WDAT2 LIN P4 CPDAT2 Tool[1]:cmttorch Base[1]:vrashatel ;%{PE}
  ;FOLD Parameters ;%{h}
    ;Params IlfProvider=kukaroboter.arctech.arcofflin; Kuka.IsGlobalPoint=False; Kuka.PointName=P4; Kuka.BlendingEnabled=False; Kuka.MoveDataName=CPDAT2; Kuka.VelocityPath=0.01; Kuka.CurrentCDSetIndex=0; Kuka.MovementParameterFieldEnabled=True; ArcTech.WdatVarName=WDAT2; ArcTech.Basic=3.4.3.1264
  ;ENDFOLD
  $BWDSTART = FALSE
  LDAT_ACT = LCPDAT2
  FDAT_ACT = FP4
  BAS(#CP_PARAMS, gArcBasVelDefinition)
  SET_CD_PARAMS (0)
  TRIGGER WHEN PATH = ArcGetPath(#ArcOffBefore, WDAT2) DELAY = 0 DO ArcMainNG(#ArcOffBeforeOffStd, WDAT2, WP4) PRIO = -1
  TRIGGER WHEN PATH = ArcGetPath(#OnTheFlyArcOff, WDAT2) DELAY = 0 DO ArcMainNG(#ArcOffMoveStd, WDAT2, WP4) PRIO = -1
  ArcMainNG(#ArcOffBeforeMoveStd, WDAT2, WP4)
  LIN XP4
  ArcMainNG(#ArcOffAfterMoveStd, WDAT2, WP4)
;ENDFOLD
   $VEL.CP = 0.080
   LIN  {X -9.010, Y 9.010, Z 19.700, A 0.000, B 0.000, C 0.000} C_DIS

;FOLD ARCON WDAT1 LIN P3 Vel=0.5 m/s CPDAT1 Tool[1]:cmttorch Base[1]:vrashatel ;%{PE}
  ;FOLD Parameters ;%{h}
    ;Params IlfProvider=kukaroboter.arctech.arconlin; Kuka.IsGlobalPoint=False; Kuka.PointName=P3; Kuka.BlendingEnabled=False; Kuka.MoveDataName=CPDAT1; Kuka.VelocityPath=0.5; Kuka.CurrentCDSetIndex=0; Kuka.MovementParameterFieldEnabled=True; ArcTech.WdatVarName=WDAT1; ArcTech.Basic=3.4.3.1264
  ;ENDFOLD
  $BWDSTART = FALSE
  LDAT_ACT = LCPDAT1
  FDAT_ACT = FP3
  BAS(#CP_PARAMS, 0.5)
  SET_CD_PARAMS (0)
  TRIGGER WHEN DISTANCE = 1 DELAY = ArcGetDelay(#PreDefinition, WDAT1) DO ArcMainNG(#PreDefinition, WDAT1, WP3) PRIO = -1
  TRIGGER WHEN PATH = ArcGetPath(#OnTheFlyArcOn, WDAT1) DELAY = ArcGetDelay(#GasPreflow, WDAT1) DO ArcMainNG(#GasPreflow, WDAT1, WP3) PRIO = -1
  TRIGGER WHEN PATH = ArcGetPath(#OnTheFlyArcOn, WDAT1) DELAY = 0 DO ArcMainNG(#ArcOnMoveStd, WDAT1, WP3) PRIO = -1
  ArcMainNG(#ArcOnBeforeMoveStd, WDAT1, WP3)
  LIN XP3
  ArcMainNG(#ArcOnAfterMoveStd, WDAT1, WP3)
;ENDFOLD
   $VEL.CP = 0.060
   LIN  {X -9.010, Y -9.010, Z 19.700, A 0.000, B 0.000, C 0.000} C_DIS
   $VEL.CP = 0.060
   LIN  {X 9.010, Y -9.010, Z 19.700, A 0.000, B 0.000, C 0.000} C_DIS
   $VEL.CP = 0.060
   LIN  {X 9.010, Y 9.010, Z 19.700, A 0.000, B 0.000, C 0.000} C_DIS
   $VEL.CP = 0.060
   LIN  {X -9.010, Y 9.010, Z 19.700, A 0.000, B 0.000, C 0.000} C_DIS

;FOLD ARCOFF WDAT2 LIN P4 CPDAT2 Tool[1]:cmttorch Base[1]:vrashatel ;%{PE}
  ;FOLD Parameters ;%{h}
    ;Params IlfProvider=kukaroboter.arctech.arcofflin; Kuka.IsGlobalPoint=False; Kuka.PointName=P4; Kuka.BlendingEnabled=False; Kuka.MoveDataName=CPDAT2; Kuka.VelocityPath=0.01; Kuka.CurrentCDSetIndex=0; Kuka.MovementParameterFieldEnabled=True; ArcTech.WdatVarName=WDAT2; ArcTech.Basic=3.4.3.1264
  ;ENDFOLD
  $BWDSTART = FALSE
  LDAT_ACT = LCPDAT2
  FDAT_ACT = FP4
  BAS(#CP_PARAMS, gArcBasVelDefinition)
  SET_CD_PARAMS (0)
  TRIGGER WHEN PATH = ArcGetPath(#ArcOffBefore, WDAT2) DELAY = 0 DO ArcMainNG(#ArcOffBeforeOffStd, WDAT2, WP4) PRIO = -1
  TRIGGER WHEN PATH = ArcGetPath(#OnTheFlyArcOff, WDAT2) DELAY = 0 DO ArcMainNG(#ArcOffMoveStd, WDAT2, WP4) PRIO = -1
  ArcMainNG(#ArcOffBeforeMoveStd, WDAT2, WP4)
  LIN XP4
  ArcMainNG(#ArcOffAfterMoveStd, WDAT2, WP4)
;ENDFOLD
   $VEL.CP = 0.080
   LIN  {X -9.290, Y 9.010, Z 19.700, A 0.000, B 0.000, C 0.000} C_DIS
   $VEL.CP = 0.080
   LIN  {X -9.218, Y 9.218, Z 19.700, A 0.000, B 0.000, C 0.000} C_DIS
   $VEL.CP = 0.080
   LIN  {X -4.304, Y 9.190, Z 19.700, A 0.000, B 0.000, C 0.000} C_DIS
   $VEL.CP = 0.080
   LIN  {X -4.304, Y 7.108, Z 19.700, A 0.000, B 0.000, C 0.000} C_DIS
   $VEL.CP = 0.080
   LIN  {X -4.584, Y 7.308, Z 19.700, A 0.000, B 0.000, C 0.000} C_DIS

;FOLD ARCON WDAT1 LIN P3 Vel=0.5 m/s CPDAT1 Tool[1]:cmttorch Base[1]:vrashatel ;%{PE}
  ;FOLD Parameters ;%{h}
    ;Params IlfProvider=kukaroboter.arctech.arconlin; Kuka.IsGlobalPoint=False; Kuka.PointName=P3; Kuka.BlendingEnabled=False; Kuka.MoveDataName=CPDAT1; Kuka.VelocityPath=0.5; Kuka.CurrentCDSetIndex=0; Kuka.MovementParameterFieldEnabled=True; ArcTech.WdatVarName=WDAT1; ArcTech.Basic=3.4.3.1264
  ;ENDFOLD
  $BWDSTART = FALSE
  LDAT_ACT = LCPDAT1
  FDAT_ACT = FP3
  BAS(#CP_PARAMS, 0.5)
  SET_CD_PARAMS (0)
  TRIGGER WHEN DISTANCE = 1 DELAY = ArcGetDelay(#PreDefinition, WDAT1) DO ArcMainNG(#PreDefinition, WDAT1, WP3) PRIO = -1
  TRIGGER WHEN PATH = ArcGetPath(#OnTheFlyArcOn, WDAT1) DELAY = ArcGetDelay(#GasPreflow, WDAT1) DO ArcMainNG(#GasPreflow, WDAT1, WP3) PRIO = -1
  TRIGGER WHEN PATH = ArcGetPath(#OnTheFlyArcOn, WDAT1) DELAY = 0 DO ArcMainNG(#ArcOnMoveStd, WDAT1, WP3) PRIO = -1
  ArcMainNG(#ArcOnBeforeMoveStd, WDAT1, WP3)
  LIN XP3
  ArcMainNG(#ArcOnAfterMoveStd, WDAT1, WP3)
;ENDFOLD
   $VEL.CP = 0.025
   LIN  {X -4.584, Y 7.308, Z 19.700, A 0.000, B 0.000, C 0.000} C_DIS
   $VEL.CP = 0.060
   LIN  {X 4.917, Y 7.308, Z 19.700, A 0.000, B 0.000, C 0.000} C_DIS
   $VEL.CP = 0.060
   LIN  {X 4.917, Y 5.660, Z 19.700, A 0.000, B 0.000, C 0.000} C_DIS
   $VEL.CP = 0.060
   LIN  {X 0.235, Y -3.490, Z 19.700, A 0.000, B 0.000, C 0.000} C_DIS
   $VEL.CP = 0.060
   LIN  {X 5.102, Y -3.490, Z 19.700, A 0.000, B 0.000, C 0.000} C_DIS
   $VEL.CP = 0.060
   LIN  {X 5.102, Y -6.983, Z 19.700, A 0.000, B 0.000, C 0.000} C_DIS
   $VEL.CP = 0.060
   LIN  {X -4.668, Y -6.983, Z 19.700, A 0.000, B 0.000, C 0.000} C_DIS
   $VEL.CP = 0.060
   LIN  {X -4.668, Y -5.335, Z 19.700, A 0.000, B 0.000, C 0.000} C_DIS
   $VEL.CP = 0.060
   LIN  {X 0.001, Y 3.815, Z 19.700, A 0.000, B 0.000, C 0.000} C_DIS
   $VEL.CP = 0.060
   LIN  {X -4.584, Y 3.815, Z 19.700, A 0.000, B 0.000, C 0.000} C_DIS
   $VEL.CP = 0.060
   LIN  {X -4.584, Y 7.308, Z 19.700, A 0.000, B 0.000, C 0.000} C_DIS

;FOLD ARCOFF WDAT2 LIN P4 CPDAT2 Tool[1]:cmttorch Base[1]:vrashatel ;%{PE}
  ;FOLD Parameters ;%{h}
    ;Params IlfProvider=kukaroboter.arctech.arcofflin; Kuka.IsGlobalPoint=False; Kuka.PointName=P4; Kuka.BlendingEnabled=False; Kuka.MoveDataName=CPDAT2; Kuka.VelocityPath=0.01; Kuka.CurrentCDSetIndex=0; Kuka.MovementParameterFieldEnabled=True; ArcTech.WdatVarName=WDAT2; ArcTech.Basic=3.4.3.1264
  ;ENDFOLD
  $BWDSTART = FALSE
  LDAT_ACT = LCPDAT2
  FDAT_ACT = FP4
  BAS(#CP_PARAMS, gArcBasVelDefinition)
  SET_CD_PARAMS (0)
  TRIGGER WHEN PATH = ArcGetPath(#ArcOffBefore, WDAT2) DELAY = 0 DO ArcMainNG(#ArcOffBeforeOffStd, WDAT2, WP4) PRIO = -1
  TRIGGER WHEN PATH = ArcGetPath(#OnTheFlyArcOff, WDAT2) DELAY = 0 DO ArcMainNG(#ArcOffMoveStd, WDAT2, WP4) PRIO = -1
  ArcMainNG(#ArcOffBeforeMoveStd, WDAT2, WP4)
  LIN XP4
  ArcMainNG(#ArcOffAfterMoveStd, WDAT2, WP4)
;ENDFOLD
   $VEL.CP = 0.080
   LIN  {X -4.304, Y 7.058, Z 19.700, A 0.000, B 0.000, C 0.000} C_DIS
   $VEL.CP = 0.080
   LIN  {X 4.723, Y 7.114, Z 19.700, A 0.000, B 0.000, C 0.000} C_DIS
   $VEL.CP = 0.080
   LIN  {X 4.723, Y 9.190, Z 19.700, A 0.000, B 0.000, C 0.000} C_DIS
   $VEL.CP = 0.080
   LIN  {X 8.706, Y 9.290, Z 19.700, A 0.000, B 0.000, C 0.000} C_DIS
   $VEL.CP = 0.080
   LIN  {X 8.706, Y 8.829, Z 19.700, A 0.000, B 0.000, C 0.000} C_DIS

;FOLD ARCON WDAT1 LIN P3 Vel=0.5 m/s CPDAT1 Tool[1]:cmttorch Base[1]:vrashatel ;%{PE}
  ;FOLD Parameters ;%{h}
    ;Params IlfProvider=kukaroboter.arctech.arconlin; Kuka.IsGlobalPoint=False; Kuka.PointName=P3; Kuka.BlendingEnabled=False; Kuka.MoveDataName=CPDAT1; Kuka.VelocityPath=0.5; Kuka.CurrentCDSetIndex=0; Kuka.MovementParameterFieldEnabled=True; ArcTech.WdatVarName=WDAT1; ArcTech.Basic=3.4.3.1264
  ;ENDFOLD
  $BWDSTART = FALSE
  LDAT_ACT = LCPDAT1
  FDAT_ACT = FP3
  BAS(#CP_PARAMS, 0.5)
  SET_CD_PARAMS (0)
  TRIGGER WHEN DISTANCE = 1 DELAY = ArcGetDelay(#PreDefinition, WDAT1) DO ArcMainNG(#PreDefinition, WDAT1, WP3) PRIO = -1
  TRIGGER WHEN PATH = ArcGetPath(#OnTheFlyArcOn, WDAT1) DELAY = ArcGetDelay(#GasPreflow, WDAT1) DO ArcMainNG(#GasPreflow, WDAT1, WP3) PRIO = -1
  TRIGGER WHEN PATH = ArcGetPath(#OnTheFlyArcOn, WDAT1) DELAY = 0 DO ArcMainNG(#ArcOnMoveStd, WDAT1, WP3) PRIO = -1
  ArcMainNG(#ArcOnBeforeMoveStd, WDAT1, WP3)
  LIN XP3
  ArcMainNG(#ArcOnAfterMoveStd, WDAT1, WP3)
;ENDFOLD
   $VEL.CP = 0.025
   LIN  {X 8.706, Y 8.829, Z 19.700, A 0.000, B 0.000, C 0.000} C_DIS
   $VEL.CP = 0.060
   LIN  {X 8.829, Y 8.706, Z 19.700, A 0.000, B 0.000, C 0.000} C_DIS

;FOLD ARCOFF WDAT2 LIN P4 CPDAT2 Tool[1]:cmttorch Base[1]:vrashatel ;%{PE}
  ;FOLD Parameters ;%{h}
    ;Params IlfProvider=kukaroboter.arctech.arcofflin; Kuka.IsGlobalPoint=False; Kuka.PointName=P4; Kuka.BlendingEnabled=False; Kuka.MoveDataName=CPDAT2; Kuka.VelocityPath=0.01; Kuka.CurrentCDSetIndex=0; Kuka.MovementParameterFieldEnabled=True; ArcTech.WdatVarName=WDAT2; ArcTech.Basic=3.4.3.1264
  ;ENDFOLD
  $BWDSTART = FALSE
  LDAT_ACT = LCPDAT2
  FDAT_ACT = FP4
  BAS(#CP_PARAMS, gArcBasVelDefinition)
  SET_CD_PARAMS (0)
  TRIGGER WHEN PATH = ArcGetPath(#ArcOffBefore, WDAT2) DELAY = 0 DO ArcMainNG(#ArcOffBeforeOffStd, WDAT2, WP4) PRIO = -1
  TRIGGER WHEN PATH = ArcGetPath(#OnTheFlyArcOff, WDAT2) DELAY = 0 DO ArcMainNG(#ArcOffMoveStd, WDAT2, WP4) PRIO = -1
  ArcMainNG(#ArcOffBeforeMoveStd, WDAT2, WP4)
  LIN XP4
  ArcMainNG(#ArcOffAfterMoveStd, WDAT2, WP4)
;ENDFOLD
   $VEL.CP = 0.080
   LIN  {X 8.829, Y 8.140, Z 19.700, A 0.000, B 0.000, C 0.000} C_DIS

;FOLD ARCON WDAT1 LIN P3 Vel=0.5 m/s CPDAT1 Tool[1]:cmttorch Base[1]:vrashatel ;%{PE}
  ;FOLD Parameters ;%{h}
    ;Params IlfProvider=kukaroboter.arctech.arconlin; Kuka.IsGlobalPoint=False; Kuka.PointName=P3; Kuka.BlendingEnabled=False; Kuka.MoveDataName=CPDAT1; Kuka.VelocityPath=0.5; Kuka.CurrentCDSetIndex=0; Kuka.MovementParameterFieldEnabled=True; ArcTech.WdatVarName=WDAT1; ArcTech.Basic=3.4.3.1264
  ;ENDFOLD
  $BWDSTART = FALSE
  LDAT_ACT = LCPDAT1
  FDAT_ACT = FP3
  BAS(#CP_PARAMS, 0.5)
  SET_CD_PARAMS (0)
  TRIGGER WHEN DISTANCE = 1 DELAY = ArcGetDelay(#PreDefinition, WDAT1) DO ArcMainNG(#PreDefinition, WDAT1, WP3) PRIO = -1
  TRIGGER WHEN PATH = ArcGetPath(#OnTheFlyArcOn, WDAT1) DELAY = ArcGetDelay(#GasPreflow, WDAT1) DO ArcMainNG(#GasPreflow, WDAT1, WP3) PRIO = -1
  TRIGGER WHEN PATH = ArcGetPath(#OnTheFlyArcOn, WDAT1) DELAY = 0 DO ArcMainNG(#ArcOnMoveStd, WDAT1, WP3) PRIO = -1
  ArcMainNG(#ArcOnBeforeMoveStd, WDAT1, WP3)
  LIN XP3
  ArcMainNG(#ArcOnAfterMoveStd, WDAT1, WP3)
;ENDFOLD
   $VEL.CP = 0.060
   LIN  {X 8.140, Y 8.829, Z 19.700, A 0.000, B 0.000, C 0.000} C_DIS

;FOLD ARCOFF WDAT2 LIN P4 CPDAT2 Tool[1]:cmttorch Base[1]:vrashatel ;%{PE}
  ;FOLD Parameters ;%{h}
    ;Params IlfProvider=kukaroboter.arctech.arcofflin; Kuka.IsGlobalPoint=False; Kuka.PointName=P4; Kuka.BlendingEnabled=False; Kuka.MoveDataName=CPDAT2; Kuka.VelocityPath=0.01; Kuka.CurrentCDSetIndex=0; Kuka.MovementParameterFieldEnabled=True; ArcTech.WdatVarName=WDAT2; ArcTech.Basic=3.4.3.1264
  ;ENDFOLD
  $BWDSTART = FALSE
  LDAT_ACT = LCPDAT2
  FDAT_ACT = FP4
  BAS(#CP_PARAMS, gArcBasVelDefinition)
  SET_CD_PARAMS (0)
  TRIGGER WHEN PATH = ArcGetPath(#ArcOffBefore, WDAT2) DELAY = 0 DO ArcMainNG(#ArcOffBeforeOffStd, WDAT2, WP4) PRIO = -1
  TRIGGER WHEN PATH = ArcGetPath(#OnTheFlyArcOff, WDAT2) DELAY = 0 DO ArcMainNG(#ArcOffMoveStd, WDAT2, WP4) PRIO = -1
  ArcMainNG(#ArcOffBeforeMoveStd, WDAT2, WP4)
  LIN XP4
  ArcMainNG(#ArcOffAfterMoveStd, WDAT2, WP4)
;ENDFOLD
   $VEL.CP = 0.080
   LIN  {X 7.575, Y 8.829, Z 19.700, A 0.000, B 0.000, C 0.000} C_DIS

;FOLD ARCON WDAT1 LIN P3 Vel=0.5 m/s CPDAT1 Tool[1]:cmttorch Base[1]:vrashatel ;%{PE}
  ;FOLD Parameters ;%{h}
    ;Params IlfProvider=kukaroboter.arctech.arconlin; Kuka.IsGlobalPoint=False; Kuka.PointName=P3; Kuka.BlendingEnabled=False; Kuka.MoveDataName=CPDAT1; Kuka.VelocityPath=0.5; Kuka.CurrentCDSetIndex=0; Kuka.MovementParameterFieldEnabled=True; ArcTech.WdatVarName=WDAT1; ArcTech.Basic=3.4.3.1264
  ;ENDFOLD
  $BWDSTART = FALSE
  LDAT_ACT = LCPDAT1
  FDAT_ACT = FP3
  BAS(#CP_PARAMS, 0.5)
  SET_CD_PARAMS (0)
  TRIGGER WHEN DISTANCE = 1 DELAY = ArcGetDelay(#PreDefinition, WDAT1) DO ArcMainNG(#PreDefinition, WDAT1, WP3) PRIO = -1
  TRIGGER WHEN PATH = ArcGetPath(#OnTheFlyArcOn, WDAT1) DELAY = ArcGetDelay(#GasPreflow, WDAT1) DO ArcMainNG(#GasPreflow, WDAT1, WP3) PRIO = -1
  TRIGGER WHEN PATH = ArcGetPath(#OnTheFlyArcOn, WDAT1) DELAY = 0 DO ArcMainNG(#ArcOnMoveStd, WDAT1, WP3) PRIO = -1
  ArcMainNG(#ArcOnBeforeMoveStd, WDAT1, WP3)
  LIN XP3
  ArcMainNG(#ArcOnAfterMoveStd, WDAT1, WP3)
;ENDFOLD
   $VEL.CP = 0.060
   LIN  {X 8.829, Y 7.575, Z 19.700, A 0.000, B 0.000, C 0.000} C_DIS

;FOLD ARCOFF WDAT2 LIN P4 CPDAT2 Tool[1]:cmttorch Base[1]:vrashatel ;%{PE}
  ;FOLD Parameters ;%{h}
    ;Params IlfProvider=kukaroboter.arctech.arcofflin; Kuka.IsGlobalPoint=False; Kuka.PointName=P4; Kuka.BlendingEnabled=False; Kuka.MoveDataName=CPDAT2; Kuka.VelocityPath=0.01; Kuka.CurrentCDSetIndex=0; Kuka.MovementParameterFieldEnabled=True; ArcTech.WdatVarName=WDAT2; ArcTech.Basic=3.4.3.1264
  ;ENDFOLD
  $BWDSTART = FALSE
  LDAT_ACT = LCPDAT2
  FDAT_ACT = FP4
  BAS(#CP_PARAMS, gArcBasVelDefinition)
  SET_CD_PARAMS (0)
  TRIGGER WHEN PATH = ArcGetPath(#ArcOffBefore, WDAT2) DELAY = 0 DO ArcMainNG(#ArcOffBeforeOffStd, WDAT2, WP4) PRIO = -1
  TRIGGER WHEN PATH = ArcGetPath(#OnTheFlyArcOff, WDAT2) DELAY = 0 DO ArcMainNG(#ArcOffMoveStd, WDAT2, WP4) PRIO = -1
  ArcMainNG(#ArcOffBeforeMoveStd, WDAT2, WP4)
  LIN XP4
  ArcMainNG(#ArcOffAfterMoveStd, WDAT2, WP4)
;ENDFOLD
   $VEL.CP = 0.080
   LIN  {X 8.829, Y 7.009, Z 19.700, A 0.000, B 0.000, C 0.000} C_DIS

;FOLD ARCON WDAT1 LIN P3 Vel=0.5 m/s CPDAT1 Tool[1]:cmttorch Base[1]:vrashatel ;%{PE}
  ;FOLD Parameters ;%{h}
    ;Params IlfProvider=kukaroboter.arctech.arconlin; Kuka.IsGlobalPoint=False; Kuka.PointName=P3; Kuka.BlendingEnabled=False; Kuka.MoveDataName=CPDAT1; Kuka.VelocityPath=0.5; Kuka.CurrentCDSetIndex=0; Kuka.MovementParameterFieldEnabled=True; ArcTech.WdatVarName=WDAT1; ArcTech.Basic=3.4.3.1264
  ;ENDFOLD
  $BWDSTART = FALSE
  LDAT_ACT = LCPDAT1
  FDAT_ACT = FP3
  BAS(#CP_PARAMS, 0.5)
  SET_CD_PARAMS (0)
  TRIGGER WHEN DISTANCE = 1 DELAY = ArcGetDelay(#PreDefinition, WDAT1) DO ArcMainNG(#PreDefinition, WDAT1, WP3) PRIO = -1
  TRIGGER WHEN PATH = ArcGetPath(#OnTheFlyArcOn, WDAT1) DELAY = ArcGetDelay(#GasPreflow, WDAT1) DO ArcMainNG(#GasPreflow, WDAT1, WP3) PRIO = -1
  TRIGGER WHEN PATH = ArcGetPath(#OnTheFlyArcOn, WDAT1) DELAY = 0 DO ArcMainNG(#ArcOnMoveStd, WDAT1, WP3) PRIO = -1
  ArcMainNG(#ArcOnBeforeMoveStd, WDAT1, WP3)
  LIN XP3
  ArcMainNG(#ArcOnAfterMoveStd, WDAT1, WP3)
;ENDFOLD
   $VEL.CP = 0.060
   LIN  {X 7.009, Y 8.829, Z 19.700, A 0.000, B 0.000, C 0.000} C_DIS

;FOLD ARCOFF WDAT2 LIN P4 CPDAT2 Tool[1]:cmttorch Base[1]:vrashatel ;%{PE}
  ;FOLD Parameters ;%{h}
    ;Params IlfProvider=kukaroboter.arctech.arcofflin; Kuka.IsGlobalPoint=False; Kuka.PointName=P4; Kuka.BlendingEnabled=False; Kuka.MoveDataName=CPDAT2; Kuka.VelocityPath=0.01; Kuka.CurrentCDSetIndex=0; Kuka.MovementParameterFieldEnabled=True; ArcTech.WdatVarName=WDAT2; ArcTech.Basic=3.4.3.1264
  ;ENDFOLD
  $BWDSTART = FALSE
  LDAT_ACT = LCPDAT2
  FDAT_ACT = FP4
  BAS(#CP_PARAMS, gArcBasVelDefinition)
  SET_CD_PARAMS (0)
  TRIGGER WHEN PATH = ArcGetPath(#ArcOffBefore, WDAT2) DELAY = 0 DO ArcMainNG(#ArcOffBeforeOffStd, WDAT2, WP4) PRIO = -1
  TRIGGER WHEN PATH = ArcGetPath(#OnTheFlyArcOff, WDAT2) DELAY = 0 DO ArcMainNG(#ArcOffMoveStd, WDAT2, WP4) PRIO = -1
  ArcMainNG(#ArcOffBeforeMoveStd, WDAT2, WP4)
  LIN XP4
  ArcMainNG(#ArcOffAfterMoveStd, WDAT2, WP4)
;ENDFOLD
   $VEL.CP = 0.080
   LIN  {X 6.443, Y 8.829, Z 19.700, A 0.000, B 0.000, C 0.000} C_DIS

;FOLD ARCON WDAT1 LIN P3 Vel=0.5 m/s CPDAT1 Tool[1]:cmttorch Base[1]:vrashatel ;%{PE}
  ;FOLD Parameters ;%{h}
    ;Params IlfProvider=kukaroboter.arctech.arconlin; Kuka.IsGlobalPoint=False; Kuka.PointName=P3; Kuka.BlendingEnabled=False; Kuka.MoveDataName=CPDAT1; Kuka.VelocityPath=0.5; Kuka.CurrentCDSetIndex=0; Kuka.MovementParameterFieldEnabled=True; ArcTech.WdatVarName=WDAT1; ArcTech.Basic=3.4.3.1264
  ;ENDFOLD
  $BWDSTART = FALSE
  LDAT_ACT = LCPDAT1
  FDAT_ACT = FP3
  BAS(#CP_PARAMS, 0.5)
  SET_CD_PARAMS (0)
  TRIGGER WHEN DISTANCE = 1 DELAY = ArcGetDelay(#PreDefinition, WDAT1) DO ArcMainNG(#PreDefinition, WDAT1, WP3) PRIO = -1
  TRIGGER WHEN PATH = ArcGetPath(#OnTheFlyArcOn, WDAT1) DELAY = ArcGetDelay(#GasPreflow, WDAT1) DO ArcMainNG(#GasPreflow, WDAT1, WP3) PRIO = -1
  TRIGGER WHEN PATH = ArcGetPath(#OnTheFlyArcOn, WDAT1) DELAY = 0 DO ArcMainNG(#ArcOnMoveStd, WDAT1, WP3) PRIO = -1
  ArcMainNG(#ArcOnBeforeMoveStd, WDAT1, WP3)
  LIN XP3
  ArcMainNG(#ArcOnAfterMoveStd, WDAT1, WP3)
;ENDFOLD
   $VEL.CP = 0.060
   LIN  {X 8.829, Y 6.443, Z 19.700, A 0.000, B 0.000, C 0.000} C_DIS

;FOLD ARCOFF WDAT2 LIN P4 CPDAT2 Tool[1]:cmttorch Base[1]:vrashatel ;%{PE}
  ;FOLD Parameters ;%{h}
    ;Params IlfProvider=kukaroboter.arctech.arcofflin; Kuka.IsGlobalPoint=False; Kuka.PointName=P4; Kuka.BlendingEnabled=False; Kuka.MoveDataName=CPDAT2; Kuka.VelocityPath=0.01; Kuka.CurrentCDSetIndex=0; Kuka.MovementParameterFieldEnabled=True; ArcTech.WdatVarName=WDAT2; ArcTech.Basic=3.4.3.1264
  ;ENDFOLD
  $BWDSTART = FALSE
  LDAT_ACT = LCPDAT2
  FDAT_ACT = FP4
  BAS(#CP_PARAMS, gArcBasVelDefinition)
  SET_CD_PARAMS (0)
  TRIGGER WHEN PATH = ArcGetPath(#ArcOffBefore, WDAT2) DELAY = 0 DO ArcMainNG(#ArcOffBeforeOffStd, WDAT2, WP4) PRIO = -1
  TRIGGER WHEN PATH = ArcGetPath(#OnTheFlyArcOff, WDAT2) DELAY = 0 DO ArcMainNG(#ArcOffMoveStd, WDAT2, WP4) PRIO = -1
  ArcMainNG(#ArcOffBeforeMoveStd, WDAT2, WP4)
  LIN XP4
  ArcMainNG(#ArcOffAfterMoveStd, WDAT2, WP4)
;ENDFOLD
   $VEL.CP = 0.080
   LIN  {X 8.829, Y 5.878, Z 19.700, A 0.000, B 0.000, C 0.000} C_DIS

;FOLD ARCON WDAT1 LIN P3 Vel=0.5 m/s CPDAT1 Tool[1]:cmttorch Base[1]:vrashatel ;%{PE}
  ;FOLD Parameters ;%{h}
    ;Params IlfProvider=kukaroboter.arctech.arconlin; Kuka.IsGlobalPoint=False; Kuka.PointName=P3; Kuka.BlendingEnabled=False; Kuka.MoveDataName=CPDAT1; Kuka.VelocityPath=0.5; Kuka.CurrentCDSetIndex=0; Kuka.MovementParameterFieldEnabled=True; ArcTech.WdatVarName=WDAT1; ArcTech.Basic=3.4.3.1264
  ;ENDFOLD
  $BWDSTART = FALSE
  LDAT_ACT = LCPDAT1
  FDAT_ACT = FP3
  BAS(#CP_PARAMS, 0.5)
  SET_CD_PARAMS (0)
  TRIGGER WHEN DISTANCE = 1 DELAY = ArcGetDelay(#PreDefinition, WDAT1) DO ArcMainNG(#PreDefinition, WDAT1, WP3) PRIO = -1
  TRIGGER WHEN PATH = ArcGetPath(#OnTheFlyArcOn, WDAT1) DELAY = ArcGetDelay(#GasPreflow, WDAT1) DO ArcMainNG(#GasPreflow, WDAT1, WP3) PRIO = -1
  TRIGGER WHEN PATH = ArcGetPath(#OnTheFlyArcOn, WDAT1) DELAY = 0 DO ArcMainNG(#ArcOnMoveStd, WDAT1, WP3) PRIO = -1
  ArcMainNG(#ArcOnBeforeMoveStd, WDAT1, WP3)
  LIN XP3
  ArcMainNG(#ArcOnAfterMoveStd, WDAT1, WP3)
;ENDFOLD
   $VEL.CP = 0.060
   LIN  {X 5.878, Y 8.829, Z 19.700, A 0.000, B 0.000, C 0.000} C_DIS

;FOLD ARCOFF WDAT2 LIN P4 CPDAT2 Tool[1]:cmttorch Base[1]:vrashatel ;%{PE}
  ;FOLD Parameters ;%{h}
    ;Params IlfProvider=kukaroboter.arctech.arcofflin; Kuka.IsGlobalPoint=False; Kuka.PointName=P4; Kuka.BlendingEnabled=False; Kuka.MoveDataName=CPDAT2; Kuka.VelocityPath=0.01; Kuka.CurrentCDSetIndex=0; Kuka.MovementParameterFieldEnabled=True; ArcTech.WdatVarName=WDAT2; ArcTech.Basic=3.4.3.1264
  ;ENDFOLD
  $BWDSTART = FALSE
  LDAT_ACT = LCPDAT2
  FDAT_ACT = FP4
  BAS(#CP_PARAMS, gArcBasVelDefinition)
  SET_CD_PARAMS (0)
  TRIGGER WHEN PATH = ArcGetPath(#ArcOffBefore, WDAT2) DELAY = 0 DO ArcMainNG(#ArcOffBeforeOffStd, WDAT2, WP4) PRIO = -1
  TRIGGER WHEN PATH = ArcGetPath(#OnTheFlyArcOff, WDAT2) DELAY = 0 DO ArcMainNG(#ArcOffMoveStd, WDAT2, WP4) PRIO = -1
  ArcMainNG(#ArcOffBeforeMoveStd, WDAT2, WP4)
  LIN XP4
  ArcMainNG(#ArcOffAfterMoveStd, WDAT2, WP4)
;ENDFOLD
   $VEL.CP = 0.080
   LIN  {X 5.312, Y 8.829, Z 19.700, A 0.000, B 0.000, C 0.000} C_DIS

;FOLD ARCON WDAT1 LIN P3 Vel=0.5 m/s CPDAT1 Tool[1]:cmttorch Base[1]:vrashatel ;%{PE}
  ;FOLD Parameters ;%{h}
    ;Params IlfProvider=kukaroboter.arctech.arconlin; Kuka.IsGlobalPoint=False; Kuka.PointName=P3; Kuka.BlendingEnabled=False; Kuka.MoveDataName=CPDAT1; Kuka.VelocityPath=0.5; Kuka.CurrentCDSetIndex=0; Kuka.MovementParameterFieldEnabled=True; ArcTech.WdatVarName=WDAT1; ArcTech.Basic=3.4.3.1264
  ;ENDFOLD
  $BWDSTART = FALSE
  LDAT_ACT = LCPDAT1
  FDAT_ACT = FP3
  BAS(#CP_PARAMS, 0.5)
  SET_CD_PARAMS (0)
  TRIGGER WHEN DISTANCE = 1 DELAY = ArcGetDelay(#PreDefinition, WDAT1) DO ArcMainNG(#PreDefinition, WDAT1, WP3) PRIO = -1
  TRIGGER WHEN PATH = ArcGetPath(#OnTheFlyArcOn, WDAT1) DELAY = ArcGetDelay(#GasPreflow, WDAT1) DO ArcMainNG(#GasPreflow, WDAT1, WP3) PRIO = -1
  TRIGGER WHEN PATH = ArcGetPath(#OnTheFlyArcOn, WDAT1) DELAY = 0 DO ArcMainNG(#ArcOnMoveStd, WDAT1, WP3) PRIO = -1
  ArcMainNG(#ArcOnBeforeMoveStd, WDAT1, WP3)
  LIN XP3
  ArcMainNG(#ArcOnAfterMoveStd, WDAT1, WP3)
;ENDFOLD
   $VEL.CP = 0.060
   LIN  {X 8.829, Y 5.312, Z 19.700, A 0.000, B 0.000, C 0.000} C_DIS

;FOLD ARCOFF WDAT2 LIN P4 CPDAT2 Tool[1]:cmttorch Base[1]:vrashatel ;%{PE}
  ;FOLD Parameters ;%{h}
    ;Params IlfProvider=kukaroboter.arctech.arcofflin; Kuka.IsGlobalPoint=False; Kuka.PointName=P4; Kuka.BlendingEnabled=False; Kuka.MoveDataName=CPDAT2; Kuka.VelocityPath=0.01; Kuka.CurrentCDSetIndex=0; Kuka.MovementParameterFieldEnabled=True; ArcTech.WdatVarName=WDAT2; ArcTech.Basic=3.4.3.1264
  ;ENDFOLD
  $BWDSTART = FALSE
  LDAT_ACT = LCPDAT2
  FDAT_ACT = FP4
  BAS(#CP_PARAMS, gArcBasVelDefinition)
  SET_CD_PARAMS (0)
  TRIGGER WHEN PATH = ArcGetPath(#ArcOffBefore, WDAT2) DELAY = 0 DO ArcMainNG(#ArcOffBeforeOffStd, WDAT2, WP4) PRIO = -1
  TRIGGER WHEN PATH = ArcGetPath(#OnTheFlyArcOff, WDAT2) DELAY = 0 DO ArcMainNG(#ArcOffMoveStd, WDAT2, WP4) PRIO = -1
  ArcMainNG(#ArcOffBeforeMoveStd, WDAT2, WP4)
  LIN XP4
  ArcMainNG(#ArcOffAfterMoveStd, WDAT2, WP4)
;ENDFOLD
   $VEL.CP = 0.080
   LIN  {X 8.829, Y 4.746, Z 19.700, A 0.000, B 0.000, C 0.000} C_DIS

;FOLD ARCON WDAT1 LIN P3 Vel=0.5 m/s CPDAT1 Tool[1]:cmttorch Base[1]:vrashatel ;%{PE}
  ;FOLD Parameters ;%{h}
    ;Params IlfProvider=kukaroboter.arctech.arconlin; Kuka.IsGlobalPoint=False; Kuka.PointName=P3; Kuka.BlendingEnabled=False; Kuka.MoveDataName=CPDAT1; Kuka.VelocityPath=0.5; Kuka.CurrentCDSetIndex=0; Kuka.MovementParameterFieldEnabled=True; ArcTech.WdatVarName=WDAT1; ArcTech.Basic=3.4.3.1264
  ;ENDFOLD
  $BWDSTART = FALSE
  LDAT_ACT = LCPDAT1
  FDAT_ACT = FP3
  BAS(#CP_PARAMS, 0.5)
  SET_CD_PARAMS (0)
  TRIGGER WHEN DISTANCE = 1 DELAY = ArcGetDelay(#PreDefinition, WDAT1) DO ArcMainNG(#PreDefinition, WDAT1, WP3) PRIO = -1
  TRIGGER WHEN PATH = ArcGetPath(#OnTheFlyArcOn, WDAT1) DELAY = ArcGetDelay(#GasPreflow, WDAT1) DO ArcMainNG(#GasPreflow, WDAT1, WP3) PRIO = -1
  TRIGGER WHEN PATH = ArcGetPath(#OnTheFlyArcOn, WDAT1) DELAY = 0 DO ArcMainNG(#ArcOnMoveStd, WDAT1, WP3) PRIO = -1
  ArcMainNG(#ArcOnBeforeMoveStd, WDAT1, WP3)
  LIN XP3
  ArcMainNG(#ArcOnAfterMoveStd, WDAT1, WP3)
;ENDFOLD
   $VEL.CP = 0.060
   LIN  {X 4.746, Y 8.829, Z 19.700, A 0.000, B 0.000, C 0.000} C_DIS

;FOLD ARCOFF WDAT2 LIN P4 CPDAT2 Tool[1]:cmttorch Base[1]:vrashatel ;%{PE}
  ;FOLD Parameters ;%{h}
    ;Params IlfProvider=kukaroboter.arctech.arcofflin; Kuka.IsGlobalPoint=False; Kuka.PointName=P4; Kuka.BlendingEnabled=False; Kuka.MoveDataName=CPDAT2; Kuka.VelocityPath=0.01; Kuka.CurrentCDSetIndex=0; Kuka.MovementParameterFieldEnabled=True; ArcTech.WdatVarName=WDAT2; ArcTech.Basic=3.4.3.1264
  ;ENDFOLD
  $BWDSTART = FALSE
  LDAT_ACT = LCPDAT2
  FDAT_ACT = FP4
  BAS(#CP_PARAMS, gArcBasVelDefinition)
  SET_CD_PARAMS (0)
  TRIGGER WHEN PATH = ArcGetPath(#ArcOffBefore, WDAT2) DELAY = 0 DO ArcMainNG(#ArcOffBeforeOffStd, WDAT2, WP4) PRIO = -1
  TRIGGER WHEN PATH = ArcGetPath(#OnTheFlyArcOff, WDAT2) DELAY = 0 DO ArcMainNG(#ArcOffMoveStd, WDAT2, WP4) PRIO = -1
  ArcMainNG(#ArcOffBeforeMoveStd, WDAT2, WP4)
  LIN XP4
  ArcMainNG(#ArcOffAfterMoveStd, WDAT2, WP4)
;ENDFOLD
   $VEL.CP = 0.080
   LIN  {X 4.181, Y 8.829, Z 19.700, A 0.000, B 0.000, C 0.000} C_DIS


END

--- ap_16.dat ---
&ACCESS RVP
&REL 15
&PARAM EDITMASK = *
&PARAM TEMPLATE = C:\KRC\Roboter\Template\ExpertVorgabe
&PARAM DISKPATH = KRC:\R1\Program
DEFDAT  ap_16
DECL E6POS XP1={X 170.668137,Y 87.8043442,Z 190.158340,A 179.701111,B 5.22395840E-06,C -5.58706188E-06,S 2,T 35,E1 0.0,E2 0.0,E3 0.0,E4 0.0,E5 0.0,E6 0.0}
DECL FDAT FP1={TOOL_NO 1,BASE_NO 1,IPO_FRAME #BASE,POINT2[] " "}
DECL PDAT PPDAT1={VEL 50.0000,ACC 50.0000,APO_DIST 500.000,APO_MODE #CDIS,GEAR_JERK 100.000,EXAX_IGN 0}
DECL MODULEPARAM_T LAST_TP_PARAMS={PARAMS[] "Kuka.PointName=P4; Kuka.FrameData.base_no=1; Kuka.FrameData.tool_no=1; Kuka.FrameData.ipo_frame=#BASE; Kuka.FrameData.point2=; Kuka.isglobalpoint=False; Kuka.MoveDataPtpName=PDAT3; Kuka.MovementDataPdat.apo_mode=#CDIS; Kuka.MovementDataPdat.apo_dist=500; Kuka.MovementData.vel=0.01; Kuka.MovementData.acc=50; Kuka.MovementData.exax_ign=0; Kuka.VelocityPtp=50; Kuka.BlendingEnabled=False; Kuka.APXEnabled=False; Kuka.CurrentCDSetIndex=0; Kuka.MoveDataName=CPDAT2; Kuka.MovementData.cb={AUX_PT {ORI #CONSIDER,E1 #CONSIDER,E2 #CONSIDER,E3 #CONSIDER,E4 #CONSIDER,E5 #CONSIDER,E6 #CONSIDER},TARGET_PT {ORI #INTERPOLATE,E1 #INTERPOLATE,E2 #INTERPOLATE,E3 #INTERPOLATE,E4 #INTERPOLATE,E5 #INTERPOLATE,E6 #INTERPOLATE}}; Kuka.MovementData.apo_fac=50; Kuka.MovementData.apo_dist=50; Kuka.MovementData.axis_acc=100; Kuka.MovementData.axis_vel=100; Kuka.MovementData.circ_typ=#BASE; Kuka.MovementData.jerk_fac=50; Kuka.MovementData.ori_typ=#VAR; Kuka.VelocityPath=0.01; ArcTech.WdatVarName=WDAT2                                                   "}
DECL E6POS XP2={X 44.5445099,Y 61.0237160,Z 5.54459429,A 179.701111,B 5.32584318E-06,C -5.64468837E-06,S 2,T 35,E1 0.0,E2 0.0,E3 0.0,E4 0.0,E5 0.0,E6 0.0}
DECL FDAT FP2={TOOL_NO 1,BASE_NO 1,IPO_FRAME #BASE,POINT2[] " "}
DECL PDAT PPDAT2={VEL 100.000,ACC 50.0000,APO_DIST 500.000,APO_MODE #CDIS,GEAR_JERK 100.000,EXAX_IGN 0}
DECL stArcDat_T WDAT1={WdatId[] "WDAT1",Strike {JobModeId[] "Job mode",StartTime 0.0,PreFlowTime 0.0,Channel1 0.0,Channel2 0.0,Channel3 0.0,Channel4 0.0,Channel5 0.0,Channel6 0.0,Channel7 0.0,Channel8 0.0,PurgeTime 0.0},Weld {JobModeId[] "Job mode",ParamSetId[] "Set1",Velocity 0.00416666688,Channel1 13.0000,Channel2 0.0,Channel3 0.0,Channel4 0.0,Channel5 0.0,Channel6 0.0,Channel7 0.0,Channel8 0.0},Weave {Pattern #Trapecoid,Length 2.00000,Amplitude 6.00000,Angle 90.0000,LeftSideDelay 0.0,RightSideDelay 0.0}}
DECL stArcDat_T WP3={WdatId[] "WP3",Info {Version 304031264},Strike {SeamName[] " ",PartName[] " ",SeamNumber 0,PartNumber 0,DesiredLength 0.0,LengthTolNeg 0.0,LengthTolPos 0.0,LengthCtrlActive FALSE}}
DECL E6POS XP3={X 17.3123798,Y 74.5600,Z -8.14224339,A 179.701111,B 5.31830847E-06,C -5.68684300E-06,S 2,T 35,E1 0.0,E2 0.0,E3 0.0,E4 0.0,E5 0.0,E6 0.0}
DECL FDAT FP3={TOOL_NO 1,BASE_NO 1,IPO_FRAME #BASE,POINT2[] " "}
DECL LDAT LCPDAT1={VEL 0.500000,ACC 50.0000,APO_DIST 50.0000,APO_FAC 50.0000,AXIS_VEL 100.000,AXIS_ACC 100.000,ORI_TYP #VAR,CIRC_TYP #BASE,JERK_FAC 50.0000,GEAR_JERK 100.000,EXAX_IGN 0,CB {AUX_PT {ORI #CONSIDER,E1 #CONSIDER,E2 #CONSIDER,E3 #CONSIDER,E4 #CONSIDER,E5 #CONSIDER,E6 #CONSIDER},TARGET_PT {ORI #INTERPOLATE,E1 #INTERPOLATE,E2 #INTERPOLATE,E3 #INTERPOLATE,E4 #INTERPOLATE,E5 #INTERPOLATE,E6 #INTERPOLATE}}}
DECL stArcDat_T WDAT2={WdatId[] "WDAT2",Crater {JobModeId[] "Job mode",ParamSetId[] "Set2",CraterTime 0.500000,PostflowTime 2.00000,Channel1 13.0000,Channel2 0.0,Channel3 0.0,Channel4 0.0,Channel5 0.0,Channel6 0.0,Channel7 0.0,Channel8 0.0,BurnBackTime 0.0}}
DECL stArcDat_T WP4={WdatId[] "WP4",Info {Version 304031264}}
DECL E6POS XP4={X 198.320389,Y 74.5600,Z -8.14224243,A 179.701111,B 5.32127115E-06,C -5.69861913E-06,S 2,T 35,E1 0.0,E2 0.0,E3 0.0,E4 0.0,E5 0.0,E6 0.0}
DECL FDAT FP4={TOOL_NO 1,BASE_NO 1,IPO_FRAME #BASE,POINT2[] " "}
DECL LDAT LCPDAT2={VEL 0.01000000,ACC 50.0000,APO_DIST 50.0000,APO_FAC 50.0000,AXIS_VEL 100.000,AXIS_ACC 100.000,ORI_TYP #VAR,CIRC_TYP #BASE,JERK_FAC 50.0000,GEAR_JERK 100.000,EXAX_IGN 0,CB {AUX_PT {ORI #CONSIDER,E1 #CONSIDER,E2 #CONSIDER,E3 #CONSIDER,E4 #CONSIDER,E5 #CONSIDER,E6 #CONSIDER},TARGET_PT {ORI #INTERPOLATE,E1 #INTERPOLATE,E2 #INTERPOLATE,E3 #INTERPOLATE,E4 #INTERPOLATE,E5 #INTERPOLATE,E6 #INTERPOLATE}}}
DECL E6POS XP5={X 182.544754,Y 74.1202316,Z 135.508194,A 179.701111,B 5.32868034E-06,C -5.65961591E-06,S 2,T 35,E1 0.0,E2 0.0,E3 0.0,E4 0.0,E5 0.0,E6 0.0}
DECL FDAT FP5={TOOL_NO 1,BASE_NO 1,IPO_FRAME #BASE,POINT2[] " "}
DECL PDAT PPDAT3={VEL 50.0000,ACC 50.0000,APO_DIST 500.000,APO_MODE #CDIS,GEAR_JERK 100.000,EXAX_IGN 0}
ENDDAT
